   1:  PR[GP1:91,1] = PR[GP1:90,1] + 33.755;
   1:  PR[GP1:91,2] = PR[GP1:90,2] + -35.847;
   1:L PR[91] 10mm/sec CNT100;
   1:  PR[GP1:91,1] = PR[GP1:90,1] + 35.129;
   1:  PR[GP1:91,2] = PR[GP1:90,2] + -34.570;
   1:L PR[91] 10mm/sec CNT100;
   1:  PR[GP1:91,1] = PR[GP1:90,1] + 42.615;
   1:  PR[GP1:91,2] = PR[GP1:90,2] + -25.553;
   1:L PR[91] 10mm/sec CNT100;
   1:  PR[GP1:91,1] = PR[GP1:90,1] + 43.534;
   1:  PR[GP1:91,2] = PR[GP1:90,2] + -23.862;
   1:L PR[91] 10mm/sec CNT100;
   1:  PR[GP1:91,1] = PR[GP1:90,1] + 48.248;
   1:  PR[GP1:91,2] = PR[GP1:90,2] + -13.184;
   1:L PR[91] 10mm/sec CNT100;
   1:  PR[GP1:91,1] = PR[GP1:90,1] + 48.569;
   1:  PR[GP1:91,2] = PR[GP1:90,2] + -11.273;
   1:L PR[91] 10mm/sec CNT100;
   1:  PR[GP1:91,1] = PR[GP1:90,1] + 50.173;
   1:  PR[GP1:91,2] = PR[GP1:90,2] + 0.271;
   1:L PR[91] 10mm/sec CNT100;
   1:  PR[GP1:91,1] = PR[GP1:90,1] + 49.858;
   1:  PR[GP1:91,2] = PR[GP1:90,2] + 2.169;
   1:L PR[91] 10mm/sec CNT100;
   1:  PR[GP1:91,1] = PR[GP1:90,1] + 48.243;
   1:  PR[GP1:91,2] = PR[GP1:90,2] + 13.754;
   1:L PR[91] 10mm/sec CNT100;
   1:  PR[GP1:91,1] = PR[GP1:90,1] + 43.532;
   1:  PR[GP1:91,2] = PR[GP1:90,2] + 24.424;
   1:L PR[91] 10mm/sec CNT100;
   1:  PR[GP1:91,1] = PR[GP1:90,1] + 42.610;
   1:  PR[GP1:91,2] = PR[GP1:90,2] + 26.118;
   1:L PR[91] 10mm/sec CNT100;
   1:  PR[GP1:91,1] = PR[GP1:90,1] + 35.124;
   1:  PR[GP1:91,2] = PR[GP1:90,2] + 35.135;
   1:L PR[91] 10mm/sec CNT100;
   1:  PR[GP1:91,1] = PR[GP1:90,1] + 33.745;
   1:  PR[GP1:91,2] = PR[GP1:90,2] + 36.412;
   1:L PR[91] 10mm/sec CNT100;
   1:  PR[GP1:91,1] = PR[GP1:90,1] + 20.382;
   1:  PR[GP1:91,2] = PR[GP1:90,2] + 44.688;
   1:L PR[91] 10mm/sec CNT100;
   1:  PR[GP1:91,1] = PR[GP1:90,1] + 18.719;
   1:  PR[GP1:91,2] = PR[GP1:90,2] + 45.443;
   1:L PR[91] 10mm/sec CNT100;
   1:  PR[GP1:91,1] = PR[GP1:90,1] + 3.168;
   1:  PR[GP1:91,2] = PR[GP1:90,2] + 48.349;
   1:L PR[91] 10mm/sec CNT100;
   1:  PR[GP1:91,1] = PR[GP1:90,1] + 1.407;
   1:  PR[GP1:91,2] = PR[GP1:90,2] + 48.537;
   1:L PR[91] 10mm/sec CNT100;
   1:  PR[GP1:91,1] = PR[GP1:90,1] + -0.266;
   1:  PR[GP1:91,2] = PR[GP1:90,2] + 48.243;
   1:L PR[91] 10mm/sec CNT100;
   1:  PR[GP1:91,1] = PR[GP1:90,1] + -1.940;
   1:  PR[GP1:91,2] = PR[GP1:90,2] + 48.537;
   1:L PR[91] 10mm/sec CNT100;
   1:  PR[GP1:91,1] = PR[GP1:90,1] + -3.702;
   1:  PR[GP1:91,2] = PR[GP1:90,2] + 48.349;
   1:L PR[91] 10mm/sec CNT100;
   1:  PR[GP1:91,1] = PR[GP1:90,1] + -19.248;
   1:  PR[GP1:91,2] = PR[GP1:90,2] + 45.442;
   1:L PR[91] 10mm/sec CNT100;
   1:  PR[GP1:91,1] = PR[GP1:90,1] + -20.911;
   1:  PR[GP1:91,2] = PR[GP1:90,2] + 44.687;
   1:L PR[91] 10mm/sec CNT100;
   1:  PR[GP1:91,1] = PR[GP1:90,1] + -34.271;
   1:  PR[GP1:91,2] = PR[GP1:90,2] + 36.412;
   1:L PR[91] 10mm/sec CNT100;
   1:  PR[GP1:91,1] = PR[GP1:90,1] + -35.649;
   1:  PR[GP1:91,2] = PR[GP1:90,2] + 35.137;
   1:L PR[91] 10mm/sec CNT100;
   1:  PR[GP1:91,1] = PR[GP1:90,1] + -43.135;
   1:  PR[GP1:91,2] = PR[GP1:90,2] + 26.120;
   1:L PR[91] 10mm/sec CNT100;
   1:  PR[GP1:91,1] = PR[GP1:90,1] + -44.058;
   1:  PR[GP1:91,2] = PR[GP1:90,2] + 24.423;
   1:L PR[91] 10mm/sec CNT100;
   1:  PR[GP1:91,1] = PR[GP1:90,1] + -48.772;
   1:  PR[GP1:91,2] = PR[GP1:90,2] + 13.745;
   1:L PR[91] 10mm/sec CNT100;
   1:  PR[GP1:91,1] = PR[GP1:90,1] + -49.096;
   1:  PR[GP1:91,2] = PR[GP1:90,2] + 11.782;
   1:L PR[91] 10mm/sec CNT100;
   1:  PR[GP1:91,1] = PR[GP1:90,1] + -50.699;
   1:  PR[GP1:91,2] = PR[GP1:90,2] + 0.287;
   1:L PR[91] 10mm/sec CNT100;
   1:  PR[GP1:91,1] = PR[GP1:90,1] + -50.386;
   1:  PR[GP1:91,2] = PR[GP1:90,2] + -1.605;
   1:L PR[91] 10mm/sec CNT100;
   1:  PR[GP1:91,1] = PR[GP1:90,1] + -48.770;
   1:  PR[GP1:91,2] = PR[GP1:90,2] + -13.190;
   1:L PR[91] 10mm/sec CNT100;
   1:  PR[GP1:91,1] = PR[GP1:90,1] + -44.059;
   1:  PR[GP1:91,2] = PR[GP1:90,2] + -23.861;
   1:L PR[91] 10mm/sec CNT100;
   1:  PR[GP1:91,1] = PR[GP1:90,1] + -43.140;
   1:  PR[GP1:91,2] = PR[GP1:90,2] + -25.555;
   1:L PR[91] 10mm/sec CNT100;
   1:  PR[GP1:91,1] = PR[GP1:90,1] + -35.654;
   1:  PR[GP1:91,2] = PR[GP1:90,2] + -34.572;
   1:L PR[91] 10mm/sec CNT100;
   1:  PR[GP1:91,1] = PR[GP1:90,1] + -34.281;
   1:  PR[GP1:91,2] = PR[GP1:90,2] + -35.848;
   1:L PR[91] 10mm/sec CNT100;
   1:  PR[GP1:91,1] = PR[GP1:90,1] + -20.921;
   1:  PR[GP1:91,2] = PR[GP1:90,2] + -44.122;
   1:L PR[91] 10mm/sec CNT100;
   1:  PR[GP1:91,1] = PR[GP1:90,1] + -19.263;
   1:  PR[GP1:91,2] = PR[GP1:90,2] + -44.880;
   1:L PR[91] 10mm/sec CNT100;
   1:  PR[GP1:91,1] = PR[GP1:90,1] + -3.717;
   1:  PR[GP1:91,2] = PR[GP1:90,2] + -47.787;
   1:L PR[91] 10mm/sec CNT100;
   1:  PR[GP1:91,1] = PR[GP1:90,1] + -1.956;
   1:  PR[GP1:91,2] = PR[GP1:90,2] + -47.980;
   1:L PR[91] 10mm/sec CNT100;
   1:  PR[GP1:91,1] = PR[GP1:90,1] + -0.266;
   1:  PR[GP1:91,2] = PR[GP1:90,2] + -47.697;
   1:L PR[91] 10mm/sec CNT100;
   1:  PR[GP1:91,1] = PR[GP1:90,1] + 1.234;
   1:  PR[GP1:91,2] = PR[GP1:90,2] + -48.109;
   1:  PR[GP1:91,3] = PR[GP1:90,3] + 123.525;
   1:L PR[91] 10mm/sec CNT100;
   1:  PR[GP1:91,1] = PR[GP1:90,1] + 2.783;
   1:  PR[GP1:91,2] = PR[GP1:90,2] + -47.939;
   1:L PR[91] 10mm/sec CNT100;
   1:  PR[GP1:91,1] = PR[GP1:90,1] + 18.608;
   1:  PR[GP1:91,2] = PR[GP1:90,2] + -44.981;
   1:L PR[91] 10mm/sec CNT100;
   1:  PR[GP1:91,1] = PR[GP1:90,1] + 20.067;
   1:  PR[GP1:91,2] = PR[GP1:90,2] + -44.315;
   1:L PR[91] 10mm/sec CNT100;
   1:  PR[GP1:91,1] = PR[GP1:90,1] + 33.677;
   1:  PR[GP1:91,2] = PR[GP1:90,2] + -35.886;
   1:L PR[91] 10mm/sec CNT100;
   1:  PR[GP1:91,1] = PR[GP1:90,1] + 34.888;
   1:  PR[GP1:91,2] = PR[GP1:90,2] + -34.760;
   1:L PR[91] 10mm/sec CNT100;
   1:  PR[GP1:91,1] = PR[GP1:90,1] + 42.517;
   1:  PR[GP1:91,2] = PR[GP1:90,2] + -25.570;
   1:L PR[91] 10mm/sec CNT100;
   1:  PR[GP1:91,1] = PR[GP1:90,1] + 43.328;
   1:  PR[GP1:91,2] = PR[GP1:90,2] + -24.078;
   1:L PR[91] 10mm/sec CNT100;
   1:  PR[GP1:91,1] = PR[GP1:90,1] + 48.135;
   1:  PR[GP1:91,2] = PR[GP1:90,2] + -13.189;
   1:L PR[91] 10mm/sec CNT100;
   1:  PR[GP1:91,1] = PR[GP1:90,1] + 48.418;
   1:  PR[GP1:91,2] = PR[GP1:90,2] + -11.503;
   1:L PR[91] 10mm/sec CNT100;
   1:  PR[GP1:91,1] = PR[GP1:90,1] + 50.055;
   1:  PR[GP1:91,2] = PR[GP1:90,2] + 0.271;
   1:L PR[91] 10mm/sec CNT100;
   1:  PR[GP1:91,1] = PR[GP1:90,1] + 49.778;
   1:  PR[GP1:91,2] = PR[GP1:90,2] + 1.945;
   1:L PR[91] 10mm/sec CNT100;
   1:  PR[GP1:91,1] = PR[GP1:90,1] + 48.130;
   1:  PR[GP1:91,2] = PR[GP1:90,2] + 13.759;
   1:L PR[91] 10mm/sec CNT100;
   1:  PR[GP1:91,1] = PR[GP1:90,1] + 43.326;
   1:  PR[GP1:91,2] = PR[GP1:90,2] + 24.640;
   1:L PR[91] 10mm/sec CNT100;
   1:  PR[GP1:91,1] = PR[GP1:90,1] + 42.512;
   1:  PR[GP1:91,2] = PR[GP1:90,2] + 26.134;
   1:L PR[91] 10mm/sec CNT100;
   1:  PR[GP1:91,1] = PR[GP1:90,1] + 34.883;
   1:  PR[GP1:91,2] = PR[GP1:90,2] + 35.324;
   1:L PR[91] 10mm/sec CNT100;
   1:  PR[GP1:91,1] = PR[GP1:90,1] + 33.668;
   1:  PR[GP1:91,2] = PR[GP1:90,2] + 36.450;
   1:L PR[91] 10mm/sec CNT100;
   1:  PR[GP1:91,1] = PR[GP1:90,1] + 20.058;
   1:  PR[GP1:91,2] = PR[GP1:90,2] + 44.879;
   1:L PR[91] 10mm/sec CNT100;
   1:  PR[GP1:91,1] = PR[GP1:90,1] + 18.595;
   1:  PR[GP1:91,2] = PR[GP1:90,2] + 45.542;
   1:L PR[91] 10mm/sec CNT100;
   1:  PR[GP1:91,1] = PR[GP1:90,1] + 2.769;
   1:  PR[GP1:91,2] = PR[GP1:90,2] + 48.500;
   1:L PR[91] 10mm/sec CNT100;
   1:  PR[GP1:91,1] = PR[GP1:90,1] + 1.220;
   1:  PR[GP1:91,2] = PR[GP1:90,2] + 48.666;
   1:L PR[91] 10mm/sec CNT100;
   1:  PR[GP1:91,1] = PR[GP1:90,1] + -0.266;
   1:  PR[GP1:91,2] = PR[GP1:90,2] + 48.405;
   1:L PR[91] 10mm/sec CNT100;
   1:  PR[GP1:91,1] = PR[GP1:90,1] + -1.753;
   1:  PR[GP1:91,2] = PR[GP1:90,2] + 48.666;
   1:L PR[91] 10mm/sec CNT100;
   1:  PR[GP1:91,1] = PR[GP1:90,1] + -3.303;
   1:  PR[GP1:91,2] = PR[GP1:90,2] + 48.501;
   1:L PR[91] 10mm/sec CNT100;
   1:  PR[GP1:91,1] = PR[GP1:90,1] + -19.124;
   1:  PR[GP1:91,2] = PR[GP1:90,2] + 45.542;
   1:L PR[91] 10mm/sec CNT100;
   1:  PR[GP1:91,1] = PR[GP1:90,1] + -20.587;
   1:  PR[GP1:91,2] = PR[GP1:90,2] + 44.877;
   1:L PR[91] 10mm/sec CNT100;
   1:  PR[GP1:91,1] = PR[GP1:90,1] + -34.193;
   1:  PR[GP1:91,2] = PR[GP1:90,2] + 36.450;
   1:L PR[91] 10mm/sec CNT100;
   1:  PR[GP1:91,1] = PR[GP1:90,1] + -35.408;
   1:  PR[GP1:91,2] = PR[GP1:90,2] + 35.326;
   1:L PR[91] 10mm/sec CNT100;
   1:  PR[GP1:91,1] = PR[GP1:90,1] + -43.038;
   1:  PR[GP1:91,2] = PR[GP1:90,2] + 26.136;
   1:L PR[91] 10mm/sec CNT100;
   1:  PR[GP1:91,1] = PR[GP1:90,1] + -43.852;
   1:  PR[GP1:91,2] = PR[GP1:90,2] + 24.639;
   1:L PR[91] 10mm/sec CNT100;
   1:  PR[GP1:91,1] = PR[GP1:90,1] + -48.659;
   1:  PR[GP1:91,2] = PR[GP1:90,2] + 13.750;
   1:L PR[91] 10mm/sec CNT100;
   1:  PR[GP1:91,1] = PR[GP1:90,1] + -48.945;
   1:  PR[GP1:91,2] = PR[GP1:90,2] + 12.018;
   1:L PR[91] 10mm/sec CNT100;
   1:  PR[GP1:91,1] = PR[GP1:90,1] + -50.581;
   1:  PR[GP1:91,2] = PR[GP1:90,2] + 0.287;
   1:L PR[91] 10mm/sec CNT100;
   1:  PR[GP1:91,1] = PR[GP1:90,1] + -50.305;
   1:  PR[GP1:91,2] = PR[GP1:90,2] + -1.382;
   1:L PR[91] 10mm/sec CNT100;
   1:  PR[GP1:91,1] = PR[GP1:90,1] + -48.657;
   1:  PR[GP1:91,2] = PR[GP1:90,2] + -13.195;
   1:L PR[91] 10mm/sec CNT100;
   1:  PR[GP1:91,1] = PR[GP1:90,1] + -43.853;
   1:  PR[GP1:91,2] = PR[GP1:90,2] + -24.077;
   1:L PR[91] 10mm/sec CNT100;
   1:  PR[GP1:91,1] = PR[GP1:90,1] + -43.043;
   1:  PR[GP1:91,2] = PR[GP1:90,2] + -25.572;
   1:L PR[91] 10mm/sec CNT100;
   1:  PR[GP1:91,1] = PR[GP1:90,1] + -35.412;
   1:  PR[GP1:91,2] = PR[GP1:90,2] + -34.763;
   1:L PR[91] 10mm/sec CNT100;
   1:  PR[GP1:91,1] = PR[GP1:90,1] + -34.202;
   1:  PR[GP1:91,2] = PR[GP1:90,2] + -35.886;
   1:L PR[91] 10mm/sec CNT100;
   1:  PR[GP1:91,1] = PR[GP1:90,1] + -20.596;
   1:  PR[GP1:91,2] = PR[GP1:90,2] + -44.313;
   1:L PR[91] 10mm/sec CNT100;
   1:  PR[GP1:91,1] = PR[GP1:90,1] + -19.137;
   1:  PR[GP1:91,2] = PR[GP1:90,2] + -44.980;
   1:L PR[91] 10mm/sec CNT100;
   1:  PR[GP1:91,1] = PR[GP1:90,1] + -3.317;
   1:  PR[GP1:91,2] = PR[GP1:90,2] + -47.939;
   1:L PR[91] 10mm/sec CNT100;
   1:  PR[GP1:91,1] = PR[GP1:90,1] + -1.767;
   1:  PR[GP1:91,2] = PR[GP1:90,2] + -48.109;
   1:L PR[91] 10mm/sec CNT100;
   1:  PR[GP1:91,1] = PR[GP1:90,1] + -0.266;
   1:  PR[GP1:91,2] = PR[GP1:90,2] + -47.857;
   1:L PR[91] 10mm/sec CNT100;
   1:  PR[GP1:91,1] = PR[GP1:90,1] + 1.044;
   1:  PR[GP1:91,2] = PR[GP1:90,2] + -48.237;
   1:  PR[GP1:91,3] = PR[GP1:90,3] + 124.135;
   1:L PR[91] 10mm/sec CNT100;
   1:  PR[GP1:91,1] = PR[GP1:90,1] + 2.382;
   1:  PR[GP1:91,2] = PR[GP1:90,2] + -48.090;
   1:L PR[91] 10mm/sec CNT100;
   1:  PR[GP1:91,1] = PR[GP1:90,1] + 18.482;
   1:  PR[GP1:91,2] = PR[GP1:90,2] + -45.081;
   1:L PR[91] 10mm/sec CNT100;
   1:  PR[GP1:91,1] = PR[GP1:90,1] + 19.742;
   1:  PR[GP1:91,2] = PR[GP1:90,2] + -44.506;
   1:L PR[91] 10mm/sec CNT100;
   1:  PR[GP1:91,1] = PR[GP1:90,1] + 33.599;
   1:  PR[GP1:91,2] = PR[GP1:90,2] + -35.924;
   1:L PR[91] 10mm/sec CNT100;
   1:  PR[GP1:91,1] = PR[GP1:90,1] + 34.646;
   1:  PR[GP1:91,2] = PR[GP1:90,2] + -34.951;
   1:L PR[91] 10mm/sec CNT100;
   1:  PR[GP1:91,1] = PR[GP1:90,1] + 42.419;
   1:  PR[GP1:91,2] = PR[GP1:90,2] + -25.586;
   1:L PR[91] 10mm/sec CNT100;
   1:  PR[GP1:91,1] = PR[GP1:90,1] + 43.121;
   1:  PR[GP1:91,2] = PR[GP1:90,2] + -24.295;
   1:L PR[91] 10mm/sec CNT100;
   1:  PR[GP1:91,1] = PR[GP1:90,1] + 48.022;
   1:  PR[GP1:91,2] = PR[GP1:90,2] + -13.194;
   1:L PR[91] 10mm/sec CNT100;
   1:  PR[GP1:91,1] = PR[GP1:90,1] + 48.267;
   1:  PR[GP1:91,2] = PR[GP1:90,2] + -11.734;
   1:L PR[91] 10mm/sec CNT100;
   1:  PR[GP1:91,1] = PR[GP1:90,1] + 49.937;
   1:  PR[GP1:91,2] = PR[GP1:90,2] + 0.271;
   1:L PR[91] 10mm/sec CNT100;
   1:  PR[GP1:91,1] = PR[GP1:90,1] + 49.697;
   1:  PR[GP1:91,2] = PR[GP1:90,2] + 1.721;
   1:L PR[91] 10mm/sec CNT100;
   1:  PR[GP1:91,1] = PR[GP1:90,1] + 48.017;
   1:  PR[GP1:91,2] = PR[GP1:90,2] + 13.763;
   1:L PR[91] 10mm/sec CNT100;
   1:  PR[GP1:91,1] = PR[GP1:90,1] + 43.120;
   1:  PR[GP1:91,2] = PR[GP1:90,2] + 24.856;
   1:L PR[91] 10mm/sec CNT100;
   1:  PR[GP1:91,1] = PR[GP1:90,1] + 42.415;
   1:  PR[GP1:91,2] = PR[GP1:90,2] + 26.149;
   1:L PR[91] 10mm/sec CNT100;
   1:  PR[GP1:91,1] = PR[GP1:90,1] + 34.642;
   1:  PR[GP1:91,2] = PR[GP1:90,2] + 35.514;
   1:L PR[91] 10mm/sec CNT100;
   1:  PR[GP1:91,1] = PR[GP1:90,1] + 33.591;
   1:  PR[GP1:91,2] = PR[GP1:90,2] + 36.487;
   1:L PR[91] 10mm/sec CNT100;
   1:  PR[GP1:91,1] = PR[GP1:90,1] + 19.734;
   1:  PR[GP1:91,2] = PR[GP1:90,2] + 45.069;
   1:L PR[91] 10mm/sec CNT100;
   1:  PR[GP1:91,1] = PR[GP1:90,1] + 18.470;
   1:  PR[GP1:91,2] = PR[GP1:90,2] + 45.642;
   1:L PR[91] 10mm/sec CNT100;
   1:  PR[GP1:91,1] = PR[GP1:90,1] + 2.371;
   1:  PR[GP1:91,2] = PR[GP1:90,2] + 48.652;
   1:L PR[91] 10mm/sec CNT100;
   1:  PR[GP1:91,1] = PR[GP1:90,1] + 1.033;
   1:  PR[GP1:91,2] = PR[GP1:90,2] + 48.795;
   1:L PR[91] 10mm/sec CNT100;
   1:  PR[GP1:91,1] = PR[GP1:90,1] + -0.266;
   1:  PR[GP1:91,2] = PR[GP1:90,2] + 48.566;
   1:L PR[91] 10mm/sec CNT100;
   1:  PR[GP1:91,1] = PR[GP1:90,1] + -1.566;
   1:  PR[GP1:91,2] = PR[GP1:90,2] + 48.794;
   1:L PR[91] 10mm/sec CNT100;
   1:  PR[GP1:91,1] = PR[GP1:90,1] + -2.905;
   1:  PR[GP1:91,2] = PR[GP1:90,2] + 48.652;
   1:L PR[91] 10mm/sec CNT100;
   1:  PR[GP1:91,1] = PR[GP1:90,1] + -19.000;
   1:  PR[GP1:91,2] = PR[GP1:90,2] + 45.641;
   1:L PR[91] 10mm/sec CNT100;
   1:  PR[GP1:91,1] = PR[GP1:90,1] + -20.263;
   1:  PR[GP1:91,2] = PR[GP1:90,2] + 45.068;
   1:L PR[91] 10mm/sec CNT100;
   1:  PR[GP1:91,1] = PR[GP1:90,1] + -34.116;
   1:  PR[GP1:91,2] = PR[GP1:90,2] + 36.488;
   1:L PR[91] 10mm/sec CNT100;
   1:  PR[GP1:91,1] = PR[GP1:90,1] + -35.166;
   1:  PR[GP1:91,2] = PR[GP1:90,2] + 35.516;
   1:L PR[91] 10mm/sec CNT100;
   1:  PR[GP1:91,1] = PR[GP1:90,1] + -42.941;
   1:  PR[GP1:91,2] = PR[GP1:90,2] + 26.151;
   1:L PR[91] 10mm/sec CNT100;
   1:  PR[GP1:91,1] = PR[GP1:90,1] + -43.646;
   1:  PR[GP1:91,2] = PR[GP1:90,2] + 24.855;
   1:L PR[91] 10mm/sec CNT100;
   1:  PR[GP1:91,1] = PR[GP1:90,1] + -48.546;
   1:  PR[GP1:91,2] = PR[GP1:90,2] + 13.755;
   1:L PR[91] 10mm/sec CNT100;
   1:  PR[GP1:91,1] = PR[GP1:90,1] + -48.794;
   1:  PR[GP1:91,2] = PR[GP1:90,2] + 12.255;
   1:L PR[91] 10mm/sec CNT100;
   1:  PR[GP1:91,1] = PR[GP1:90,1] + -50.463;
   1:  PR[GP1:91,2] = PR[GP1:90,2] + 0.287;
   1:L PR[91] 10mm/sec CNT100;
   1:  PR[GP1:91,1] = PR[GP1:90,1] + -50.224;
   1:  PR[GP1:91,2] = PR[GP1:90,2] + -1.158;
   1:L PR[91] 10mm/sec CNT100;
   1:  PR[GP1:91,1] = PR[GP1:90,1] + -48.544;
   1:  PR[GP1:91,2] = PR[GP1:90,2] + -13.201;
   1:L PR[91] 10mm/sec CNT100;
   1:  PR[GP1:91,1] = PR[GP1:90,1] + -43.647;
   1:  PR[GP1:91,2] = PR[GP1:90,2] + -24.294;
   1:L PR[91] 10mm/sec CNT100;
   1:  PR[GP1:91,1] = PR[GP1:90,1] + -42.945;
   1:  PR[GP1:91,2] = PR[GP1:90,2] + -25.588;
   1:L PR[91] 10mm/sec CNT100;
   1:  PR[GP1:91,1] = PR[GP1:90,1] + -35.170;
   1:  PR[GP1:91,2] = PR[GP1:90,2] + -34.953;
   1:L PR[91] 10mm/sec CNT100;
   1:  PR[GP1:91,1] = PR[GP1:90,1] + -34.124;
   1:  PR[GP1:91,2] = PR[GP1:90,2] + -35.925;
   1:L PR[91] 10mm/sec CNT100;
   1:  PR[GP1:91,1] = PR[GP1:90,1] + -20.271;
   1:  PR[GP1:91,2] = PR[GP1:90,2] + -44.505;
   1:L PR[91] 10mm/sec CNT100;
   1:  PR[GP1:91,1] = PR[GP1:90,1] + -19.011;
   1:  PR[GP1:91,2] = PR[GP1:90,2] + -45.080;
   1:L PR[91] 10mm/sec CNT100;
   1:  PR[GP1:91,1] = PR[GP1:90,1] + -2.916;
   1:  PR[GP1:91,2] = PR[GP1:90,2] + -48.090;
   1:L PR[91] 10mm/sec CNT100;
   1:  PR[GP1:91,1] = PR[GP1:90,1] + -1.578;
   1:  PR[GP1:91,2] = PR[GP1:90,2] + -48.237;
   1:L PR[91] 10mm/sec CNT100;
   1:  PR[GP1:91,1] = PR[GP1:90,1] + -0.266;
   1:  PR[GP1:91,2] = PR[GP1:90,2] + -48.017;
   1:L PR[91] 10mm/sec CNT100;
   1:  PR[GP1:91,1] = PR[GP1:90,1] + 0.855;
   1:  PR[GP1:91,2] = PR[GP1:90,2] + -48.366;
   1:  PR[GP1:91,3] = PR[GP1:90,3] + 124.745;
   1:L PR[91] 10mm/sec CNT100;
   1:  PR[GP1:91,1] = PR[GP1:90,1] + 1.982;
   1:  PR[GP1:91,2] = PR[GP1:90,2] + -48.242;
   1:L PR[91] 10mm/sec CNT100;
   1:  PR[GP1:91,1] = PR[GP1:90,1] + 18.355;
   1:  PR[GP1:91,2] = PR[GP1:90,2] + -45.182;
   1:L PR[91] 10mm/sec CNT100;
   1:  PR[GP1:91,1] = PR[GP1:90,1] + 19.416;
   1:  PR[GP1:91,2] = PR[GP1:90,2] + -44.697;
   1:L PR[91] 10mm/sec CNT100;
   1:  PR[GP1:91,1] = PR[GP1:90,1] + 33.520;
   1:  PR[GP1:91,2] = PR[GP1:90,2] + -35.962;
   1:L PR[91] 10mm/sec CNT100;
   1:  PR[GP1:91,1] = PR[GP1:90,1] + 34.404;
   1:  PR[GP1:91,2] = PR[GP1:90,2] + -35.141;
   1:L PR[91] 10mm/sec CNT100;
   1:  PR[GP1:91,1] = PR[GP1:90,1] + 42.321;
   1:  PR[GP1:91,2] = PR[GP1:90,2] + -25.603;
   1:L PR[91] 10mm/sec CNT100;
   1:  PR[GP1:91,1] = PR[GP1:90,1] + 42.915;
   1:  PR[GP1:91,2] = PR[GP1:90,2] + -24.511;
   1:L PR[91] 10mm/sec CNT100;
   1:  PR[GP1:91,1] = PR[GP1:90,1] + 47.909;
   1:  PR[GP1:91,2] = PR[GP1:90,2] + -13.199;
   1:L PR[91] 10mm/sec CNT100;
   1:  PR[GP1:91,1] = PR[GP1:90,1] + 48.116;
   1:  PR[GP1:91,2] = PR[GP1:90,2] + -11.965;
   1:L PR[91] 10mm/sec CNT100;
   1:  PR[GP1:91,1] = PR[GP1:90,1] + 49.819;
   1:  PR[GP1:91,2] = PR[GP1:90,2] + 0.271;
   1:L PR[91] 10mm/sec CNT100;
   1:  PR[GP1:91,1] = PR[GP1:90,1] + 49.616;
   1:  PR[GP1:91,2] = PR[GP1:90,2] + 1.497;
   1:L PR[91] 10mm/sec CNT100;
   1:  PR[GP1:91,1] = PR[GP1:90,1] + 47.904;
   1:  PR[GP1:91,2] = PR[GP1:90,2] + 13.768;
   1:L PR[91] 10mm/sec CNT100;
   1:  PR[GP1:91,1] = PR[GP1:90,1] + 42.914;
   1:  PR[GP1:91,2] = PR[GP1:90,2] + 25.071;
   1:L PR[91] 10mm/sec CNT100;
   1:  PR[GP1:91,1] = PR[GP1:90,1] + 42.318;
   1:  PR[GP1:91,2] = PR[GP1:90,2] + 26.165;
   1:L PR[91] 10mm/sec CNT100;
   1:  PR[GP1:91,1] = PR[GP1:90,1] + 34.400;
   1:  PR[GP1:91,2] = PR[GP1:90,2] + 35.703;
   1:L PR[91] 10mm/sec CNT100;
   1:  PR[GP1:91,1] = PR[GP1:90,1] + 33.514;
   1:  PR[GP1:91,2] = PR[GP1:90,2] + 36.525;
   1:L PR[91] 10mm/sec CNT100;
   1:  PR[GP1:91,1] = PR[GP1:90,1] + 19.410;
   1:  PR[GP1:91,2] = PR[GP1:90,2] + 45.260;
   1:L PR[91] 10mm/sec CNT100;
   1:  PR[GP1:91,1] = PR[GP1:90,1] + 18.346;
   1:  PR[GP1:91,2] = PR[GP1:90,2] + 45.742;
   1:L PR[91] 10mm/sec CNT100;
   1:  PR[GP1:91,1] = PR[GP1:90,1] + 1.972;
   1:  PR[GP1:91,2] = PR[GP1:90,2] + 48.803;
   1:L PR[91] 10mm/sec CNT100;
   1:  PR[GP1:91,1] = PR[GP1:90,1] + 0.845;
   1:  PR[GP1:91,2] = PR[GP1:90,2] + 48.923;
   1:L PR[91] 10mm/sec CNT100;
   1:  PR[GP1:91,1] = PR[GP1:90,1] + -0.266;
   1:  PR[GP1:91,2] = PR[GP1:90,2] + 48.728;
   1:L PR[91] 10mm/sec CNT100;
   1:  PR[GP1:91,1] = PR[GP1:90,1] + -1.379;
   1:  PR[GP1:91,2] = PR[GP1:90,2] + 48.923;
   1:L PR[91] 10mm/sec CNT100;
   1:  PR[GP1:91,1] = PR[GP1:90,1] + -2.506;
   1:  PR[GP1:91,2] = PR[GP1:90,2] + 48.803;
   1:L PR[91] 10mm/sec CNT100;
   1:  PR[GP1:91,1] = PR[GP1:90,1] + -18.875;
   1:  PR[GP1:91,2] = PR[GP1:90,2] + 45.741;
   1:L PR[91] 10mm/sec CNT100;
   1:  PR[GP1:91,1] = PR[GP1:90,1] + -19.939;
   1:  PR[GP1:91,2] = PR[GP1:90,2] + 45.258;
   1:L PR[91] 10mm/sec CNT100;
   1:  PR[GP1:91,1] = PR[GP1:90,1] + -34.039;
   1:  PR[GP1:91,2] = PR[GP1:90,2] + 36.525;
   1:L PR[91] 10mm/sec CNT100;
   1:  PR[GP1:91,1] = PR[GP1:90,1] + -34.925;
   1:  PR[GP1:91,2] = PR[GP1:90,2] + 35.705;
   1:L PR[91] 10mm/sec CNT100;
   1:  PR[GP1:91,1] = PR[GP1:90,1] + -42.844;
   1:  PR[GP1:91,2] = PR[GP1:90,2] + 26.167;
   1:L PR[91] 10mm/sec CNT100;
   1:  PR[GP1:91,1] = PR[GP1:90,1] + -43.440;
   1:  PR[GP1:91,2] = PR[GP1:90,2] + 25.071;
   1:L PR[91] 10mm/sec CNT100;
   1:  PR[GP1:91,1] = PR[GP1:90,1] + -48.434;
   1:  PR[GP1:91,2] = PR[GP1:90,2] + 13.760;
   1:L PR[91] 10mm/sec CNT100;
   1:  PR[GP1:91,1] = PR[GP1:90,1] + -48.643;
   1:  PR[GP1:91,2] = PR[GP1:90,2] + 12.491;
   1:L PR[91] 10mm/sec CNT100;
   1:  PR[GP1:91,1] = PR[GP1:90,1] + -50.345;
   1:  PR[GP1:91,2] = PR[GP1:90,2] + 0.287;
   1:L PR[91] 10mm/sec CNT100;
   1:  PR[GP1:91,1] = PR[GP1:90,1] + -50.143;
   1:  PR[GP1:91,2] = PR[GP1:90,2] + -0.935;
   1:L PR[91] 10mm/sec CNT100;
   1:  PR[GP1:91,1] = PR[GP1:90,1] + -48.431;
   1:  PR[GP1:91,2] = PR[GP1:90,2] + -13.206;
   1:L PR[91] 10mm/sec CNT100;
   1:  PR[GP1:91,1] = PR[GP1:90,1] + -43.441;
   1:  PR[GP1:91,2] = PR[GP1:90,2] + -24.511;
   1:L PR[91] 10mm/sec CNT100;
   1:  PR[GP1:91,1] = PR[GP1:90,1] + -42.847;
   1:  PR[GP1:91,2] = PR[GP1:90,2] + -25.605;
   1:L PR[91] 10mm/sec CNT100;
   1:  PR[GP1:91,1] = PR[GP1:90,1] + -34.928;
   1:  PR[GP1:91,2] = PR[GP1:90,2] + -35.143;
   1:L PR[91] 10mm/sec CNT100;
   1:  PR[GP1:91,1] = PR[GP1:90,1] + -34.045;
   1:  PR[GP1:91,2] = PR[GP1:90,2] + -35.963;
   1:L PR[91] 10mm/sec CNT100;
   1:  PR[GP1:91,1] = PR[GP1:90,1] + -19.945;
   1:  PR[GP1:91,2] = PR[GP1:90,2] + -44.696;
   1:L PR[91] 10mm/sec CNT100;
   1:  PR[GP1:91,1] = PR[GP1:90,1] + -18.885;
   1:  PR[GP1:91,2] = PR[GP1:90,2] + -45.181;
   1:L PR[91] 10mm/sec CNT100;
   1:  PR[GP1:91,1] = PR[GP1:90,1] + -2.516;
   1:  PR[GP1:91,2] = PR[GP1:90,2] + -48.242;
   1:L PR[91] 10mm/sec CNT100;
   1:  PR[GP1:91,1] = PR[GP1:90,1] + -1.389;
   1:  PR[GP1:91,2] = PR[GP1:90,2] + -48.366;
   1:L PR[91] 10mm/sec CNT100;
   1:  PR[GP1:91,1] = PR[GP1:90,1] + -0.266;
   1:  PR[GP1:91,2] = PR[GP1:90,2] + -48.178;
   1:L PR[91] 10mm/sec CNT100;
   1:  PR[GP1:91,1] = PR[GP1:90,1] + 0.666;
   1:  PR[GP1:91,2] = PR[GP1:90,2] + -48.494;
   1:  PR[GP1:91,3] = PR[GP1:90,3] + 125.355;
   1:L PR[91] 10mm/sec CNT100;
   1:  PR[GP1:91,1] = PR[GP1:90,1] + 1.581;
   1:  PR[GP1:91,2] = PR[GP1:90,2] + -48.394;
   1:L PR[91] 10mm/sec CNT100;
   1:  PR[GP1:91,1] = PR[GP1:90,1] + 18.229;
   1:  PR[GP1:91,2] = PR[GP1:90,2] + -45.282;
   1:L PR[91] 10mm/sec CNT100;
   1:  PR[GP1:91,1] = PR[GP1:90,1] + 19.091;
   1:  PR[GP1:91,2] = PR[GP1:90,2] + -44.889;
   1:L PR[91] 10mm/sec CNT100;
   1:  PR[GP1:91,1] = PR[GP1:90,1] + 33.442;
   1:  PR[GP1:91,2] = PR[GP1:90,2] + -36.001;
   1:L PR[91] 10mm/sec CNT100;
   1:  PR[GP1:91,1] = PR[GP1:90,1] + 34.162;
   1:  PR[GP1:91,2] = PR[GP1:90,2] + -35.331;
   1:L PR[91] 10mm/sec CNT100;
   1:  PR[GP1:91,1] = PR[GP1:90,1] + 42.224;
   1:  PR[GP1:91,2] = PR[GP1:90,2] + -25.620;
   1:L PR[91] 10mm/sec CNT100;
   1:  PR[GP1:91,1] = PR[GP1:90,1] + 42.709;
   1:  PR[GP1:91,2] = PR[GP1:90,2] + -24.727;
   1:L PR[91] 10mm/sec CNT100;
   1:  PR[GP1:91,1] = PR[GP1:90,1] + 47.796;
   1:  PR[GP1:91,2] = PR[GP1:90,2] + -13.204;
   1:L PR[91] 10mm/sec CNT100;
   1:  PR[GP1:91,1] = PR[GP1:90,1] + 47.965;
   1:  PR[GP1:91,2] = PR[GP1:90,2] + -12.195;
   1:L PR[91] 10mm/sec CNT100;
   1:  PR[GP1:91,1] = PR[GP1:90,1] + 49.701;
   1:  PR[GP1:91,2] = PR[GP1:90,2] + 0.271;
   1:L PR[91] 10mm/sec CNT100;
   1:  PR[GP1:91,1] = PR[GP1:90,1] + 49.535;
   1:  PR[GP1:91,2] = PR[GP1:90,2] + 1.273;
   1:L PR[91] 10mm/sec CNT100;
   1:  PR[GP1:91,1] = PR[GP1:90,1] + 47.792;
   1:  PR[GP1:91,2] = PR[GP1:90,2] + 13.772;
   1:L PR[91] 10mm/sec CNT100;
   1:  PR[GP1:91,1] = PR[GP1:90,1] + 42.708;
   1:  PR[GP1:91,2] = PR[GP1:90,2] + 25.287;
   1:L PR[91] 10mm/sec CNT100;
   1:  PR[GP1:91,1] = PR[GP1:90,1] + 42.221;
   1:  PR[GP1:91,2] = PR[GP1:90,2] + 26.181;
   1:L PR[91] 10mm/sec CNT100;
   1:  PR[GP1:91,1] = PR[GP1:90,1] + 34.159;
   1:  PR[GP1:91,2] = PR[GP1:90,2] + 35.893;
   1:L PR[91] 10mm/sec CNT100;
   1:  PR[GP1:91,1] = PR[GP1:90,1] + 33.437;
   1:  PR[GP1:91,2] = PR[GP1:90,2] + 36.562;
   1:L PR[91] 10mm/sec CNT100;
   1:  PR[GP1:91,1] = PR[GP1:90,1] + 19.086;
   1:  PR[GP1:91,2] = PR[GP1:90,2] + 45.450;
   1:L PR[91] 10mm/sec CNT100;
   1:  PR[GP1:91,1] = PR[GP1:90,1] + 18.221;
   1:  PR[GP1:91,2] = PR[GP1:90,2] + 45.842;
   1:L PR[91] 10mm/sec CNT100;
   1:  PR[GP1:91,1] = PR[GP1:90,1] + 1.573;
   1:  PR[GP1:91,2] = PR[GP1:90,2] + 48.954;
   1:L PR[91] 10mm/sec CNT100;
   1:  PR[GP1:91,1] = PR[GP1:90,1] + 0.658;
   1:  PR[GP1:91,2] = PR[GP1:90,2] + 49.052;
   1:L PR[91] 10mm/sec CNT100;
   1:  PR[GP1:91,1] = PR[GP1:90,1] + -0.266;
   1:  PR[GP1:91,2] = PR[GP1:90,2] + 48.889;
   1:L PR[91] 10mm/sec CNT100;
   1:  PR[GP1:91,1] = PR[GP1:90,1] + -1.192;
   1:  PR[GP1:91,2] = PR[GP1:90,2] + 49.052;
   1:L PR[91] 10mm/sec CNT100;
   1:  PR[GP1:91,1] = PR[GP1:90,1] + -2.108;
   1:  PR[GP1:91,2] = PR[GP1:90,2] + 48.954;
   1:L PR[91] 10mm/sec CNT100;
   1:  PR[GP1:91,1] = PR[GP1:90,1] + -18.751;
   1:  PR[GP1:91,2] = PR[GP1:90,2] + 45.841;
   1:L PR[91] 10mm/sec CNT100;
   1:  PR[GP1:91,1] = PR[GP1:90,1] + -19.615;
   1:  PR[GP1:91,2] = PR[GP1:90,2] + 45.449;
   1:L PR[91] 10mm/sec CNT100;
   1:  PR[GP1:91,1] = PR[GP1:90,1] + -33.962;
   1:  PR[GP1:91,2] = PR[GP1:90,2] + 36.563;
   1:L PR[91] 10mm/sec CNT100;
   1:  PR[GP1:91,1] = PR[GP1:90,1] + -34.684;
   1:  PR[GP1:91,2] = PR[GP1:90,2] + 35.895;
   1:L PR[91] 10mm/sec CNT100;
   1:  PR[GP1:91,1] = PR[GP1:90,1] + -42.747;
   1:  PR[GP1:91,2] = PR[GP1:90,2] + 26.183;
   1:L PR[91] 10mm/sec CNT100;
   1:  PR[GP1:91,1] = PR[GP1:90,1] + -43.234;
   1:  PR[GP1:91,2] = PR[GP1:90,2] + 25.287;
   1:L PR[91] 10mm/sec CNT100;
   1:  PR[GP1:91,1] = PR[GP1:90,1] + -48.321;
   1:  PR[GP1:91,2] = PR[GP1:90,2] + 13.765;
   1:L PR[91] 10mm/sec CNT100;
   1:  PR[GP1:91,1] = PR[GP1:90,1] + -48.492;
   1:  PR[GP1:91,2] = PR[GP1:90,2] + 12.727;
   1:L PR[91] 10mm/sec CNT100;
   1:  PR[GP1:91,1] = PR[GP1:90,1] + -50.227;
   1:  PR[GP1:91,2] = PR[GP1:90,2] + 0.287;
   1:L PR[91] 10mm/sec CNT100;
   1:  PR[GP1:91,1] = PR[GP1:90,1] + -50.062;
   1:  PR[GP1:91,2] = PR[GP1:90,2] + -0.711;
   1:L PR[91] 10mm/sec CNT100;
   1:  PR[GP1:91,1] = PR[GP1:90,1] + -48.319;
   1:  PR[GP1:91,2] = PR[GP1:90,2] + -13.211;
   1:L PR[91] 10mm/sec CNT100;
   1:  PR[GP1:91,1] = PR[GP1:90,1] + -43.235;
   1:  PR[GP1:91,2] = PR[GP1:90,2] + -24.727;
   1:L PR[91] 10mm/sec CNT100;
   1:  PR[GP1:91,1] = PR[GP1:90,1] + -42.749;
   1:  PR[GP1:91,2] = PR[GP1:90,2] + -25.621;
   1:L PR[91] 10mm/sec CNT100;
   1:  PR[GP1:91,1] = PR[GP1:90,1] + -34.686;
   1:  PR[GP1:91,2] = PR[GP1:90,2] + -35.333;
   1:L PR[91] 10mm/sec CNT100;
   1:  PR[GP1:91,1] = PR[GP1:90,1] + -33.967;
   1:  PR[GP1:91,2] = PR[GP1:90,2] + -36.001;
   1:L PR[91] 10mm/sec CNT100;
   1:  PR[GP1:91,1] = PR[GP1:90,1] + -19.620;
   1:  PR[GP1:91,2] = PR[GP1:90,2] + -44.887;
   1:L PR[91] 10mm/sec CNT100;
   1:  PR[GP1:91,1] = PR[GP1:90,1] + -18.758;
   1:  PR[GP1:91,2] = PR[GP1:90,2] + -45.281;
   1:L PR[91] 10mm/sec CNT100;
   1:  PR[GP1:91,1] = PR[GP1:90,1] + -2.116;
   1:  PR[GP1:91,2] = PR[GP1:90,2] + -48.394;
   1:L PR[91] 10mm/sec CNT100;
   1:  PR[GP1:91,1] = PR[GP1:90,1] + -1.200;
   1:  PR[GP1:91,2] = PR[GP1:90,2] + -48.494;
   1:L PR[91] 10mm/sec CNT100;
   1:  PR[GP1:91,1] = PR[GP1:90,1] + -0.266;
   1:  PR[GP1:91,2] = PR[GP1:90,2] + -48.338;
   1:L PR[91] 10mm/sec CNT100;
   1:  PR[GP1:91,1] = PR[GP1:90,1] + 0.476;
   1:  PR[GP1:91,2] = PR[GP1:90,2] + -48.623;
   1:  PR[GP1:91,3] = PR[GP1:90,3] + 125.965;
   1:L PR[91] 10mm/sec CNT100;
   1:  PR[GP1:91,1] = PR[GP1:90,1] + 1.181;
   1:  PR[GP1:91,2] = PR[GP1:90,2] + -48.545;
   1:L PR[91] 10mm/sec CNT100;
   1:  PR[GP1:91,1] = PR[GP1:90,1] + 18.103;
   1:  PR[GP1:91,2] = PR[GP1:90,2] + -45.382;
   1:L PR[91] 10mm/sec CNT100;
   1:  PR[GP1:91,1] = PR[GP1:90,1] + 18.765;
   1:  PR[GP1:91,2] = PR[GP1:90,2] + -45.080;
   1:L PR[91] 10mm/sec CNT100;
   1:  PR[GP1:91,1] = PR[GP1:90,1] + 33.363;
   1:  PR[GP1:91,2] = PR[GP1:90,2] + -36.039;
   1:L PR[91] 10mm/sec CNT100;
   1:  PR[GP1:91,1] = PR[GP1:90,1] + 33.920;
   1:  PR[GP1:91,2] = PR[GP1:90,2] + -35.522;
   1:L PR[91] 10mm/sec CNT100;
   1:  PR[GP1:91,1] = PR[GP1:90,1] + 42.126;
   1:  PR[GP1:91,2] = PR[GP1:90,2] + -25.636;
   1:L PR[91] 10mm/sec CNT100;
   1:  PR[GP1:91,1] = PR[GP1:90,1] + 42.503;
   1:  PR[GP1:91,2] = PR[GP1:90,2] + -24.943;
   1:L PR[91] 10mm/sec CNT100;
   1:  PR[GP1:91,1] = PR[GP1:90,1] + 47.683;
   1:  PR[GP1:91,2] = PR[GP1:90,2] + -13.209;
   1:L PR[91] 10mm/sec CNT100;
   1:  PR[GP1:91,1] = PR[GP1:90,1] + 47.814;
   1:  PR[GP1:91,2] = PR[GP1:90,2] + -12.426;
   1:L PR[91] 10mm/sec CNT100;
   1:  PR[GP1:91,1] = PR[GP1:90,1] + 49.583;
   1:  PR[GP1:91,2] = PR[GP1:90,2] + 0.271;
   1:L PR[91] 10mm/sec CNT100;
   1:  PR[GP1:91,1] = PR[GP1:90,1] + 49.454;
   1:  PR[GP1:91,2] = PR[GP1:90,2] + 1.048;
   1:L PR[91] 10mm/sec CNT100;
   1:  PR[GP1:91,1] = PR[GP1:90,1] + 47.679;
   1:  PR[GP1:91,2] = PR[GP1:90,2] + 13.777;
   1:L PR[91] 10mm/sec CNT100;
   1:  PR[GP1:91,1] = PR[GP1:90,1] + 42.502;
   1:  PR[GP1:91,2] = PR[GP1:90,2] + 25.503;
   1:L PR[91] 10mm/sec CNT100;
   1:  PR[GP1:91,1] = PR[GP1:90,1] + 42.124;
   1:  PR[GP1:91,2] = PR[GP1:90,2] + 26.197;
   1:L PR[91] 10mm/sec CNT100;
   1:  PR[GP1:91,1] = PR[GP1:90,1] + 33.918;
   1:  PR[GP1:91,2] = PR[GP1:90,2] + 36.082;
   1:L PR[91] 10mm/sec CNT100;
   1:  PR[GP1:91,1] = PR[GP1:90,1] + 33.359;
   1:  PR[GP1:91,2] = PR[GP1:90,2] + 36.600;
   1:L PR[91] 10mm/sec CNT100;
   1:  PR[GP1:91,1] = PR[GP1:90,1] + 18.761;
   1:  PR[GP1:91,2] = PR[GP1:90,2] + 45.641;
   1:L PR[91] 10mm/sec CNT100;
   1:  PR[GP1:91,1] = PR[GP1:90,1] + 18.097;
   1:  PR[GP1:91,2] = PR[GP1:90,2] + 45.942;
   1:L PR[91] 10mm/sec CNT100;
   1:  PR[GP1:91,1] = PR[GP1:90,1] + 1.175;
   1:  PR[GP1:91,2] = PR[GP1:90,2] + 49.105;
   1:L PR[91] 10mm/sec CNT100;
   1:  PR[GP1:91,1] = PR[GP1:90,1] + 0.471;
   1:  PR[GP1:91,2] = PR[GP1:90,2] + 49.180;
   1:L PR[91] 10mm/sec CNT100;
   1:  PR[GP1:91,1] = PR[GP1:90,1] + -0.267;
   1:  PR[GP1:91,2] = PR[GP1:90,2] + 49.050;
   1:L PR[91] 10mm/sec CNT100;
   1:  PR[GP1:91,1] = PR[GP1:90,1] + -1.005;
   1:  PR[GP1:91,2] = PR[GP1:90,2] + 49.180;
   1:L PR[91] 10mm/sec CNT100;
   1:  PR[GP1:91,1] = PR[GP1:90,1] + -1.709;
   1:  PR[GP1:91,2] = PR[GP1:90,2] + 49.105;
   1:L PR[91] 10mm/sec CNT100;
   1:  PR[GP1:91,1] = PR[GP1:90,1] + -18.626;
   1:  PR[GP1:91,2] = PR[GP1:90,2] + 45.941;
   1:L PR[91] 10mm/sec CNT100;
   1:  PR[GP1:91,1] = PR[GP1:90,1] + -19.291;
   1:  PR[GP1:91,2] = PR[GP1:90,2] + 45.639;
   1:L PR[91] 10mm/sec CNT100;
   1:  PR[GP1:91,1] = PR[GP1:90,1] + -33.885;
   1:  PR[GP1:91,2] = PR[GP1:90,2] + 36.600;
   1:L PR[91] 10mm/sec CNT100;
   1:  PR[GP1:91,1] = PR[GP1:90,1] + -34.442;
   1:  PR[GP1:91,2] = PR[GP1:90,2] + 36.084;
   1:L PR[91] 10mm/sec CNT100;
   1:  PR[GP1:91,1] = PR[GP1:90,1] + -42.650;
   1:  PR[GP1:91,2] = PR[GP1:90,2] + 26.198;
   1:L PR[91] 10mm/sec CNT100;
   1:  PR[GP1:91,1] = PR[GP1:90,1] + -43.028;
   1:  PR[GP1:91,2] = PR[GP1:90,2] + 25.503;
   1:L PR[91] 10mm/sec CNT100;
   1:  PR[GP1:91,1] = PR[GP1:90,1] + -48.208;
   1:  PR[GP1:91,2] = PR[GP1:90,2] + 13.769;
   1:L PR[91] 10mm/sec CNT100;
   1:  PR[GP1:91,1] = PR[GP1:90,1] + -48.341;
   1:  PR[GP1:91,2] = PR[GP1:90,2] + 12.964;
   1:L PR[91] 10mm/sec CNT100;
   1:  PR[GP1:91,1] = PR[GP1:90,1] + -50.109;
   1:  PR[GP1:91,2] = PR[GP1:90,2] + 0.287;
   1:L PR[91] 10mm/sec CNT100;
   1:  PR[GP1:91,1] = PR[GP1:90,1] + -49.981;
   1:  PR[GP1:91,2] = PR[GP1:90,2] + -0.488;
   1:L PR[91] 10mm/sec CNT100;
   1:  PR[GP1:91,1] = PR[GP1:90,1] + -48.206;
   1:  PR[GP1:91,2] = PR[GP1:90,2] + -13.217;
   1:L PR[91] 10mm/sec CNT100;
   1:  PR[GP1:91,1] = PR[GP1:90,1] + -43.028;
   1:  PR[GP1:91,2] = PR[GP1:90,2] + -24.944;
   1:L PR[91] 10mm/sec CNT100;
   1:  PR[GP1:91,1] = PR[GP1:90,1] + -42.652;
   1:  PR[GP1:91,2] = PR[GP1:90,2] + -25.638;
   1:L PR[91] 10mm/sec CNT100;
   1:  PR[GP1:91,1] = PR[GP1:90,1] + -34.445;
   1:  PR[GP1:91,2] = PR[GP1:90,2] + -35.524;
   1:L PR[91] 10mm/sec CNT100;
   1:  PR[GP1:91,1] = PR[GP1:90,1] + -33.889;
   1:  PR[GP1:91,2] = PR[GP1:90,2] + -36.040;
   1:L PR[91] 10mm/sec CNT100;
   1:  PR[GP1:91,1] = PR[GP1:90,1] + -19.295;
   1:  PR[GP1:91,2] = PR[GP1:90,2] + -45.079;
   1:L PR[91] 10mm/sec CNT100;
   1:  PR[GP1:91,1] = PR[GP1:90,1] + -18.632;
   1:  PR[GP1:91,2] = PR[GP1:90,2] + -45.381;
   1:L PR[91] 10mm/sec CNT100;
   1:  PR[GP1:91,1] = PR[GP1:90,1] + -1.715;
   1:  PR[GP1:91,2] = PR[GP1:90,2] + -48.545;
   1:L PR[91] 10mm/sec CNT100;
   1:  PR[GP1:91,1] = PR[GP1:90,1] + -1.010;
   1:  PR[GP1:91,2] = PR[GP1:90,2] + -48.623;
   1:L PR[91] 10mm/sec CNT100;
   1:  PR[GP1:91,1] = PR[GP1:90,1] + -0.267;
   1:  PR[GP1:91,2] = PR[GP1:90,2] + -48.498;
   1:L PR[91] 10mm/sec CNT100;
   1:  PR[GP1:91,1] = PR[GP1:90,1] + 0.287;
   1:  PR[GP1:91,2] = PR[GP1:90,2] + -48.751;
   1:  PR[GP1:91,3] = PR[GP1:90,3] + 126.575;
   1:L PR[91] 10mm/sec CNT100;
   1:  PR[GP1:91,1] = PR[GP1:90,1] + 0.780;
   1:  PR[GP1:91,2] = PR[GP1:90,2] + -48.697;
   1:L PR[91] 10mm/sec CNT100;
   1:  PR[GP1:91,1] = PR[GP1:90,1] + 17.977;
   1:  PR[GP1:91,2] = PR[GP1:90,2] + -45.483;
   1:L PR[91] 10mm/sec CNT100;
   1:  PR[GP1:91,1] = PR[GP1:90,1] + 18.440;
   1:  PR[GP1:91,2] = PR[GP1:90,2] + -45.271;
   1:L PR[91] 10mm/sec CNT100;
   1:  PR[GP1:91,1] = PR[GP1:90,1] + 33.285;
   1:  PR[GP1:91,2] = PR[GP1:90,2] + -36.077;
   1:L PR[91] 10mm/sec CNT100;
   1:  PR[GP1:91,1] = PR[GP1:90,1] + 33.678;
   1:  PR[GP1:91,2] = PR[GP1:90,2] + -35.712;
   1:L PR[91] 10mm/sec CNT100;
   1:  PR[GP1:91,1] = PR[GP1:90,1] + 42.028;
   1:  PR[GP1:91,2] = PR[GP1:90,2] + -25.653;
   1:L PR[91] 10mm/sec CNT100;
   1:  PR[GP1:91,1] = PR[GP1:90,1] + 42.296;
   1:  PR[GP1:91,2] = PR[GP1:90,2] + -25.160;
   1:L PR[91] 10mm/sec CNT100;
   1:  PR[GP1:91,1] = PR[GP1:90,1] + 47.570;
   1:  PR[GP1:91,2] = PR[GP1:90,2] + -13.214;
   1:L PR[91] 10mm/sec CNT100;
   1:  PR[GP1:91,1] = PR[GP1:90,1] + 47.664;
   1:  PR[GP1:91,2] = PR[GP1:90,2] + -12.657;
   1:L PR[91] 10mm/sec CNT100;
   1:  PR[GP1:91,1] = PR[GP1:90,1] + 49.465;
   1:  PR[GP1:91,2] = PR[GP1:90,2] + 0.271;
   1:L PR[91] 10mm/sec CNT100;
   1:  PR[GP1:91,1] = PR[GP1:90,1] + 49.373;
   1:  PR[GP1:91,2] = PR[GP1:90,2] + 0.824;
   1:L PR[91] 10mm/sec CNT100;
   1:  PR[GP1:91,1] = PR[GP1:90,1] + 47.566;
   1:  PR[GP1:91,2] = PR[GP1:90,2] + 13.781;
   1:L PR[91] 10mm/sec CNT100;
   1:  PR[GP1:91,1] = PR[GP1:90,1] + 42.296;
   1:  PR[GP1:91,2] = PR[GP1:90,2] + 25.719;
   1:L PR[91] 10mm/sec CNT100;
   1:  PR[GP1:91,1] = PR[GP1:90,1] + 42.027;
   1:  PR[GP1:91,2] = PR[GP1:90,2] + 26.213;
   1:L PR[91] 10mm/sec CNT100;
   1:  PR[GP1:91,1] = PR[GP1:90,1] + 33.676;
   1:  PR[GP1:91,2] = PR[GP1:90,2] + 36.272;
   1:L PR[91] 10mm/sec CNT100;
   1:  PR[GP1:91,1] = PR[GP1:90,1] + 33.282;
   1:  PR[GP1:91,2] = PR[GP1:90,2] + 36.637;
   1:L PR[91] 10mm/sec CNT100;
   1:  PR[GP1:91,1] = PR[GP1:90,1] + 18.437;
   1:  PR[GP1:91,2] = PR[GP1:90,2] + 45.831;
   1:L PR[91] 10mm/sec CNT100;
   1:  PR[GP1:91,1] = PR[GP1:90,1] + 17.972;
   1:  PR[GP1:91,2] = PR[GP1:90,2] + 46.042;
   1:L PR[91] 10mm/sec CNT100;
   1:  PR[GP1:91,1] = PR[GP1:90,1] + 0.776;
   1:  PR[GP1:91,2] = PR[GP1:90,2] + 49.256;
   1:L PR[91] 10mm/sec CNT100;
   1:  PR[GP1:91,1] = PR[GP1:90,1] + 0.284;
   1:  PR[GP1:91,2] = PR[GP1:90,2] + 49.309;
   1:L PR[91] 10mm/sec CNT100;
   1:  PR[GP1:91,1] = PR[GP1:90,1] + -0.267;
   1:  PR[GP1:91,2] = PR[GP1:90,2] + 49.212;
   1:L PR[91] 10mm/sec CNT100;
   1:  PR[GP1:91,1] = PR[GP1:90,1] + -0.818;
   1:  PR[GP1:91,2] = PR[GP1:90,2] + 49.309;
   1:L PR[91] 10mm/sec CNT100;
   1:  PR[GP1:91,1] = PR[GP1:90,1] + -1.311;
   1:  PR[GP1:91,2] = PR[GP1:90,2] + 49.256;
   1:L PR[91] 10mm/sec CNT100;
   1:  PR[GP1:91,1] = PR[GP1:90,1] + -18.502;
   1:  PR[GP1:91,2] = PR[GP1:90,2] + 46.041;
   1:L PR[91] 10mm/sec CNT100;
   1:  PR[GP1:91,1] = PR[GP1:90,1] + -18.967;
   1:  PR[GP1:91,2] = PR[GP1:90,2] + 45.830;
   1:L PR[91] 10mm/sec CNT100;
   1:  PR[GP1:91,1] = PR[GP1:90,1] + -33.807;
   1:  PR[GP1:91,2] = PR[GP1:90,2] + 36.638;
   1:L PR[91] 10mm/sec CNT100;
   1:  PR[GP1:91,1] = PR[GP1:90,1] + -34.201;
   1:  PR[GP1:91,2] = PR[GP1:90,2] + 36.274;
   1:L PR[91] 10mm/sec CNT100;
   1:  PR[GP1:91,1] = PR[GP1:90,1] + -42.553;
   1:  PR[GP1:91,2] = PR[GP1:90,2] + 26.214;
   1:L PR[91] 10mm/sec CNT100;
   1:  PR[GP1:91,1] = PR[GP1:90,1] + -42.822;
   1:  PR[GP1:91,2] = PR[GP1:90,2] + 25.719;
   1:L PR[91] 10mm/sec CNT100;
   1:  PR[GP1:91,1] = PR[GP1:90,1] + -48.095;
   1:  PR[GP1:91,2] = PR[GP1:90,2] + 13.774;
   1:L PR[91] 10mm/sec CNT100;
   1:  PR[GP1:91,1] = PR[GP1:90,1] + -48.190;
   1:  PR[GP1:91,2] = PR[GP1:90,2] + 13.200;
   1:L PR[91] 10mm/sec CNT100;
   1:  PR[GP1:91,1] = PR[GP1:90,1] + -49.991;
   1:  PR[GP1:91,2] = PR[GP1:90,2] + 0.287;
   1:L PR[91] 10mm/sec CNT100;
   1:  PR[GP1:91,1] = PR[GP1:90,1] + -49.900;
   1:  PR[GP1:91,2] = PR[GP1:90,2] + -0.264;
   1:L PR[91] 10mm/sec CNT100;
   1:  PR[GP1:91,1] = PR[GP1:90,1] + -48.093;
   1:  PR[GP1:91,2] = PR[GP1:90,2] + -13.222;
   1:L PR[91] 10mm/sec CNT100;
   1:  PR[GP1:91,1] = PR[GP1:90,1] + -42.822;
   1:  PR[GP1:91,2] = PR[GP1:90,2] + -25.160;
   1:L PR[91] 10mm/sec CNT100;
   1:  PR[GP1:91,1] = PR[GP1:90,1] + -42.554;
   1:  PR[GP1:91,2] = PR[GP1:90,2] + -25.654;
   1:L PR[91] 10mm/sec CNT100;
   1:  PR[GP1:91,1] = PR[GP1:90,1] + -34.203;
   1:  PR[GP1:91,2] = PR[GP1:90,2] + -35.714;
   1:L PR[91] 10mm/sec CNT100;
   1:  PR[GP1:91,1] = PR[GP1:90,1] + -33.810;
   1:  PR[GP1:91,2] = PR[GP1:90,2] + -36.078;
   1:L PR[91] 10mm/sec CNT100;
   1:  PR[GP1:91,1] = PR[GP1:90,1] + -18.969;
   1:  PR[GP1:91,2] = PR[GP1:90,2] + -45.270;
   1:L PR[91] 10mm/sec CNT100;
   1:  PR[GP1:91,1] = PR[GP1:90,1] + -18.506;
   1:  PR[GP1:91,2] = PR[GP1:90,2] + -45.482;
   1:L PR[91] 10mm/sec CNT100;
   1:  PR[GP1:91,1] = PR[GP1:90,1] + -1.315;
   1:  PR[GP1:91,2] = PR[GP1:90,2] + -48.697;
   1:L PR[91] 10mm/sec CNT100;
   1:  PR[GP1:91,1] = PR[GP1:90,1] + -0.821;
   1:  PR[GP1:91,2] = PR[GP1:90,2] + -48.751;
   1:L PR[91] 10mm/sec CNT100;
   1:  PR[GP1:91,1] = PR[GP1:90,1] + -0.267;
   1:  PR[GP1:91,2] = PR[GP1:90,2] + -48.658;
   1:L PR[91] 10mm/sec CNT100;
   1:  PR[GP1:91,1] = PR[GP1:90,1] + 0.097;
   1:  PR[GP1:91,2] = PR[GP1:90,2] + -48.880;
   1:  PR[GP1:91,3] = PR[GP1:90,3] + 127.185;
   1:L PR[91] 10mm/sec CNT100;
   1:  PR[GP1:91,1] = PR[GP1:90,1] + 0.380;
   1:  PR[GP1:91,2] = PR[GP1:90,2] + -48.849;
   1:L PR[91] 10mm/sec CNT100;
   1:  PR[GP1:91,1] = PR[GP1:90,1] + 17.850;
   1:  PR[GP1:91,2] = PR[GP1:90,2] + -45.583;
   1:L PR[91] 10mm/sec CNT100;
   1:  PR[GP1:91,1] = PR[GP1:90,1] + 18.115;
   1:  PR[GP1:91,2] = PR[GP1:90,2] + -45.462;
   1:L PR[91] 10mm/sec CNT100;
   1:  PR[GP1:91,1] = PR[GP1:90,1] + 33.207;
   1:  PR[GP1:91,2] = PR[GP1:90,2] + -36.115;
   1:L PR[91] 10mm/sec CNT100;
   1:  PR[GP1:91,1] = PR[GP1:90,1] + 33.436;
   1:  PR[GP1:91,2] = PR[GP1:90,2] + -35.902;
   1:L PR[91] 10mm/sec CNT100;
   1:  PR[GP1:91,1] = PR[GP1:90,1] + 41.931;
   1:  PR[GP1:91,2] = PR[GP1:90,2] + -25.669;
   1:L PR[91] 10mm/sec CNT100;
   1:  PR[GP1:91,1] = PR[GP1:90,1] + 42.090;
   1:  PR[GP1:91,2] = PR[GP1:90,2] + -25.376;
   1:L PR[91] 10mm/sec CNT100;
   1:  PR[GP1:91,1] = PR[GP1:90,1] + 47.457;
   1:  PR[GP1:91,2] = PR[GP1:90,2] + -13.219;
   1:L PR[91] 10mm/sec CNT100;
   1:  PR[GP1:91,1] = PR[GP1:90,1] + 47.513;
   1:  PR[GP1:91,2] = PR[GP1:90,2] + -12.887;
   1:L PR[91] 10mm/sec CNT100;
   1:  PR[GP1:91,1] = PR[GP1:90,1] + 49.347;
   1:  PR[GP1:91,2] = PR[GP1:90,2] + 0.271;
   1:L PR[91] 10mm/sec CNT100;
   1:  PR[GP1:91,1] = PR[GP1:90,1] + 49.292;
   1:  PR[GP1:91,2] = PR[GP1:90,2] + 0.600;
   1:L PR[91] 10mm/sec CNT100;
   1:  PR[GP1:91,1] = PR[GP1:90,1] + 47.453;
   1:  PR[GP1:91,2] = PR[GP1:90,2] + 13.786;
   1:L PR[91] 10mm/sec CNT100;
   1:  PR[GP1:91,1] = PR[GP1:90,1] + 42.090;
   1:  PR[GP1:91,2] = PR[GP1:90,2] + 25.935;
   1:L PR[91] 10mm/sec CNT100;
   1:  PR[GP1:91,1] = PR[GP1:90,1] + 41.930;
   1:  PR[GP1:91,2] = PR[GP1:90,2] + 26.229;
   1:L PR[91] 10mm/sec CNT100;
   1:  PR[GP1:91,1] = PR[GP1:90,1] + 33.435;
   1:  PR[GP1:91,2] = PR[GP1:90,2] + 36.461;
   1:L PR[91] 10mm/sec CNT100;
   1:  PR[GP1:91,1] = PR[GP1:90,1] + 33.205;
   1:  PR[GP1:91,2] = PR[GP1:90,2] + 36.675;
   1:L PR[91] 10mm/sec CNT100;
   1:  PR[GP1:91,1] = PR[GP1:90,1] + 18.113;
   1:  PR[GP1:91,2] = PR[GP1:90,2] + 46.022;
   1:L PR[91] 10mm/sec CNT100;
   1:  PR[GP1:91,1] = PR[GP1:90,1] + 17.848;
   1:  PR[GP1:91,2] = PR[GP1:90,2] + 46.142;
   1:L PR[91] 10mm/sec CNT100;
   1:  PR[GP1:91,1] = PR[GP1:90,1] + 0.377;
   1:  PR[GP1:91,2] = PR[GP1:90,2] + 49.407;
   1:L PR[91] 10mm/sec CNT100;
   1:  PR[GP1:91,1] = PR[GP1:90,1] + 0.097;
   1:  PR[GP1:91,2] = PR[GP1:90,2] + 49.437;
   1:L PR[91] 10mm/sec CNT100;
   1:  PR[GP1:91,1] = PR[GP1:90,1] + -0.267;
   1:  PR[GP1:91,2] = PR[GP1:90,2] + 49.373;
   1:L PR[91] 10mm/sec CNT100;
   1:  PR[GP1:91,1] = PR[GP1:90,1] + -0.631;
   1:  PR[GP1:91,2] = PR[GP1:90,2] + 49.437;
   1:L PR[91] 10mm/sec CNT100;
   1:  PR[GP1:91,1] = PR[GP1:90,1] + -0.912;
   1:  PR[GP1:91,2] = PR[GP1:90,2] + 49.407;
   1:L PR[91] 10mm/sec CNT100;
   1:  PR[GP1:91,1] = PR[GP1:90,1] + -18.377;
   1:  PR[GP1:91,2] = PR[GP1:90,2] + 46.141;
   1:L PR[91] 10mm/sec CNT100;
   1:  PR[GP1:91,1] = PR[GP1:90,1] + -18.642;
   1:  PR[GP1:91,2] = PR[GP1:90,2] + 46.020;
   1:L PR[91] 10mm/sec CNT100;
   1:  PR[GP1:91,1] = PR[GP1:90,1] + -33.730;
   1:  PR[GP1:91,2] = PR[GP1:90,2] + 36.676;
   1:L PR[91] 10mm/sec CNT100;
   1:  PR[GP1:91,1] = PR[GP1:90,1] + -33.960;
   1:  PR[GP1:91,2] = PR[GP1:90,2] + 36.463;
   1:L PR[91] 10mm/sec CNT100;
   1:  PR[GP1:91,1] = PR[GP1:90,1] + -42.455;
   1:  PR[GP1:91,2] = PR[GP1:90,2] + 26.230;
   1:L PR[91] 10mm/sec CNT100;
   1:  PR[GP1:91,1] = PR[GP1:90,1] + -42.616;
   1:  PR[GP1:91,2] = PR[GP1:90,2] + 25.935;
   1:L PR[91] 10mm/sec CNT100;
   1:  PR[GP1:91,1] = PR[GP1:90,1] + -47.982;
   1:  PR[GP1:91,2] = PR[GP1:90,2] + 13.779;
   1:L PR[91] 10mm/sec CNT100;
   1:  PR[GP1:91,1] = PR[GP1:90,1] + -48.039;
   1:  PR[GP1:91,2] = PR[GP1:90,2] + 13.436;
   1:L PR[91] 10mm/sec CNT100;
   1:  PR[GP1:91,1] = PR[GP1:90,1] + -49.873;
   1:  PR[GP1:91,2] = PR[GP1:90,2] + 0.287;
   1:L PR[91] 10mm/sec CNT100;
   1:  PR[GP1:91,1] = PR[GP1:90,1] + -49.819;
   1:  PR[GP1:91,2] = PR[GP1:90,2] + -0.041;
   1:L PR[91] 10mm/sec CNT100;
   1:  PR[GP1:91,1] = PR[GP1:90,1] + -47.980;
   1:  PR[GP1:91,2] = PR[GP1:90,2] + -13.227;
   1:L PR[91] 10mm/sec CNT100;
   1:  PR[GP1:91,1] = PR[GP1:90,1] + -42.616;
   1:  PR[GP1:91,2] = PR[GP1:90,2] + -25.377;
   1:L PR[91] 10mm/sec CNT100;
   1:  PR[GP1:91,1] = PR[GP1:90,1] + -42.456;
   1:  PR[GP1:91,2] = PR[GP1:90,2] + -25.671;
   1:L PR[91] 10mm/sec CNT100;
   1:  PR[GP1:91,1] = PR[GP1:90,1] + -33.961;
   1:  PR[GP1:91,2] = PR[GP1:90,2] + -35.904;
   1:L PR[91] 10mm/sec CNT100;
   1:  PR[GP1:91,1] = PR[GP1:90,1] + -33.732;
   1:  PR[GP1:91,2] = PR[GP1:90,2] + -36.116;
   1:L PR[91] 10mm/sec CNT100;
   1:  PR[GP1:91,1] = PR[GP1:90,1] + -18.644;
   1:  PR[GP1:91,2] = PR[GP1:90,2] + -45.461;
   1:L PR[91] 10mm/sec CNT100;
   1:  PR[GP1:91,1] = PR[GP1:90,1] + -18.380;
   1:  PR[GP1:91,2] = PR[GP1:90,2] + -45.582;
   1:L PR[91] 10mm/sec CNT100;
   1:  PR[GP1:91,1] = PR[GP1:90,1] + -0.914;
   1:  PR[GP1:91,2] = PR[GP1:90,2] + -48.849;
   1:L PR[91] 10mm/sec CNT100;
   1:  PR[GP1:91,1] = PR[GP1:90,1] + -0.632;
   1:  PR[GP1:91,2] = PR[GP1:90,2] + -48.880;
   1:L PR[91] 10mm/sec CNT100;
   1:  PR[GP1:91,1] = PR[GP1:90,1] + -0.267;
   1:  PR[GP1:91,2] = PR[GP1:90,2] + -48.818;
   1:L PR[91] 10mm/sec CNT100;
   1:  PR[GP1:91,1] = PR[GP1:90,1] + -0.092;
   1:  PR[GP1:91,2] = PR[GP1:90,2] + -49.008;
   1:  PR[GP1:91,3] = PR[GP1:90,3] + 127.795;
   1:L PR[91] 10mm/sec CNT100;
   1:  PR[GP1:91,1] = PR[GP1:90,1] + -0.021;
   1:  PR[GP1:91,2] = PR[GP1:90,2] + -49.000;
   1:L PR[91] 10mm/sec CNT100;
   1:  PR[GP1:91,1] = PR[GP1:90,1] + 17.724;
   1:  PR[GP1:91,2] = PR[GP1:90,2] + -45.684;
   1:L PR[91] 10mm/sec CNT100;
   1:  PR[GP1:91,1] = PR[GP1:90,1] + 17.789;
   1:  PR[GP1:91,2] = PR[GP1:90,2] + -45.654;
   1:L PR[91] 10mm/sec CNT100;
   1:  PR[GP1:91,1] = PR[GP1:90,1] + 33.128;
   1:  PR[GP1:91,2] = PR[GP1:90,2] + -36.154;
   1:L PR[91] 10mm/sec CNT100;
   1:  PR[GP1:91,1] = PR[GP1:90,1] + 33.194;
   1:  PR[GP1:91,2] = PR[GP1:90,2] + -36.093;
   1:L PR[91] 10mm/sec CNT100;
   1:  PR[GP1:91,1] = PR[GP1:90,1] + 41.833;
   1:  PR[GP1:91,2] = PR[GP1:90,2] + -25.686;
   1:L PR[91] 10mm/sec CNT100;
   1:  PR[GP1:91,1] = PR[GP1:90,1] + 41.884;
   1:  PR[GP1:91,2] = PR[GP1:90,2] + -25.592;
   1:L PR[91] 10mm/sec CNT100;
   1:  PR[GP1:91,1] = PR[GP1:90,1] + 47.340;
   1:  PR[GP1:91,2] = PR[GP1:90,2] + -13.232;
   1:L PR[91] 10mm/sec CNT100;
   1:  PR[GP1:91,1] = PR[GP1:90,1] + 49.230;
   1:  PR[GP1:91,2] = PR[GP1:90,2] + 0.279;
   1:L PR[91] 10mm/sec CNT100;
   1:  PR[GP1:91,1] = PR[GP1:90,1] + 47.340;
   1:  PR[GP1:91,2] = PR[GP1:90,2] + 13.790;
   1:L PR[91] 10mm/sec CNT100;
   1:  PR[GP1:91,1] = PR[GP1:90,1] + 41.884;
   1:  PR[GP1:91,2] = PR[GP1:90,2] + 26.150;
   1:L PR[91] 10mm/sec CNT100;
   1:  PR[GP1:91,1] = PR[GP1:90,1] + 41.833;
   1:  PR[GP1:91,2] = PR[GP1:90,2] + 26.244;
   1:L PR[91] 10mm/sec CNT100;
   1:  PR[GP1:91,1] = PR[GP1:90,1] + 33.194;
   1:  PR[GP1:91,2] = PR[GP1:90,2] + 36.651;
   1:L PR[91] 10mm/sec CNT100;
   1:  PR[GP1:91,1] = PR[GP1:90,1] + 33.128;
   1:  PR[GP1:91,2] = PR[GP1:90,2] + 36.712;
   1:L PR[91] 10mm/sec CNT100;
   1:  PR[GP1:91,1] = PR[GP1:90,1] + 17.789;
   1:  PR[GP1:91,2] = PR[GP1:90,2] + 46.212;
   1:L PR[91] 10mm/sec CNT100;
   1:  PR[GP1:91,1] = PR[GP1:90,1] + 17.723;
   1:  PR[GP1:91,2] = PR[GP1:90,2] + 46.242;
   1:L PR[91] 10mm/sec CNT100;
   1:  PR[GP1:91,1] = PR[GP1:90,1] + -0.021;
   1:  PR[GP1:91,2] = PR[GP1:90,2] + 49.559;
   1:L PR[91] 10mm/sec CNT100;
   1:  PR[GP1:91,1] = PR[GP1:90,1] + -0.090;
   1:  PR[GP1:91,2] = PR[GP1:90,2] + 49.566;
   1:L PR[91] 10mm/sec CNT100;
   1:  PR[GP1:91,1] = PR[GP1:90,1] + -0.267;
   1:  PR[GP1:91,2] = PR[GP1:90,2] + 49.535;
   1:L PR[91] 10mm/sec CNT100;
   1:  PR[GP1:91,1] = PR[GP1:90,1] + -0.444;
   1:  PR[GP1:91,2] = PR[GP1:90,2] + 49.566;
   1:L PR[91] 10mm/sec CNT100;
   1:  PR[GP1:91,1] = PR[GP1:90,1] + -0.513;
   1:  PR[GP1:91,2] = PR[GP1:90,2] + 49.559;
   1:L PR[91] 10mm/sec CNT100;
   1:  PR[GP1:91,1] = PR[GP1:90,1] + -18.253;
   1:  PR[GP1:91,2] = PR[GP1:90,2] + 46.241;
   1:L PR[91] 10mm/sec CNT100;
   1:  PR[GP1:91,1] = PR[GP1:90,1] + -18.318;
   1:  PR[GP1:91,2] = PR[GP1:90,2] + 46.211;
   1:L PR[91] 10mm/sec CNT100;
   1:  PR[GP1:91,1] = PR[GP1:90,1] + -33.653;
   1:  PR[GP1:91,2] = PR[GP1:90,2] + 36.713;
   1:L PR[91] 10mm/sec CNT100;
   1:  PR[GP1:91,1] = PR[GP1:90,1] + -33.718;
   1:  PR[GP1:91,2] = PR[GP1:90,2] + 36.653;
   1:L PR[91] 10mm/sec CNT100;
   1:  PR[GP1:91,1] = PR[GP1:90,1] + -42.358;
   1:  PR[GP1:91,2] = PR[GP1:90,2] + 26.246;
   1:L PR[91] 10mm/sec CNT100;
   1:  PR[GP1:91,1] = PR[GP1:90,1] + -42.410;
   1:  PR[GP1:91,2] = PR[GP1:90,2] + 26.151;
   1:L PR[91] 10mm/sec CNT100;
   1:  PR[GP1:91,1] = PR[GP1:90,1] + -47.870;
   1:  PR[GP1:91,2] = PR[GP1:90,2] + 13.784;
   1:L PR[91] 10mm/sec CNT100;
   1:  PR[GP1:91,1] = PR[GP1:90,1] + -47.888;
   1:  PR[GP1:91,2] = PR[GP1:90,2] + 13.673;
   1:L PR[91] 10mm/sec CNT100;
   1:  PR[GP1:91,1] = PR[GP1:90,1] + -49.756;
   1:  PR[GP1:91,2] = PR[GP1:90,2] + 0.279;
   1:L PR[91] 10mm/sec CNT100;
   1:  PR[GP1:91,1] = PR[GP1:90,1] + -47.867;
   1:  PR[GP1:91,2] = PR[GP1:90,2] + -13.232;
   1:L PR[91] 10mm/sec CNT100;
   1:  PR[GP1:91,1] = PR[GP1:90,1] + -42.410;
   1:  PR[GP1:91,2] = PR[GP1:90,2] + -25.593;
   1:L PR[91] 10mm/sec CNT100;
   1:  PR[GP1:91,1] = PR[GP1:90,1] + -42.359;
   1:  PR[GP1:91,2] = PR[GP1:90,2] + -25.687;
   1:L PR[91] 10mm/sec CNT100;
   1:  PR[GP1:91,1] = PR[GP1:90,1] + -33.719;
   1:  PR[GP1:91,2] = PR[GP1:90,2] + -36.094;
   1:L PR[91] 10mm/sec CNT100;
   1:  PR[GP1:91,1] = PR[GP1:90,1] + -33.654;
   1:  PR[GP1:91,2] = PR[GP1:90,2] + -36.155;
   1:L PR[91] 10mm/sec CNT100;
   1:  PR[GP1:91,1] = PR[GP1:90,1] + -18.319;
   1:  PR[GP1:91,2] = PR[GP1:90,2] + -45.653;
   1:L PR[91] 10mm/sec CNT100;
   1:  PR[GP1:91,1] = PR[GP1:90,1] + -18.254;
   1:  PR[GP1:91,2] = PR[GP1:90,2] + -45.682;
   1:L PR[91] 10mm/sec CNT100;
   1:  PR[GP1:91,1] = PR[GP1:90,1] + -0.514;
   1:  PR[GP1:91,2] = PR[GP1:90,2] + -49.000;
   1:L PR[91] 10mm/sec CNT100;
   1:  PR[GP1:91,1] = PR[GP1:90,1] + -0.443;
   1:  PR[GP1:91,2] = PR[GP1:90,2] + -49.008;
   1:L PR[91] 10mm/sec CNT100;
   1:  PR[GP1:91,1] = PR[GP1:90,1] + -0.267;
   1:  PR[GP1:91,2] = PR[GP1:90,2] + -48.979;
   1:L PR[91] 10mm/sec CNT100;
   1:  PR[GP1:91,1] = PR[GP1:90,1] + 17.591;
   1:  PR[GP1:91,2] = PR[GP1:90,2] + -45.770;
   1:  PR[GP1:91,3] = PR[GP1:90,3] + 128.405;
   1:L PR[91] 10mm/sec CNT100;
   1:  PR[GP1:91,1] = PR[GP1:90,1] + 33.046;
   1:  PR[GP1:91,2] = PR[GP1:90,2] + -36.191;
   1:L PR[91] 10mm/sec CNT100;
   1:  PR[GP1:91,1] = PR[GP1:90,1] + 41.697;
   1:  PR[GP1:91,2] = PR[GP1:90,2] + -25.769;
   1:L PR[91] 10mm/sec CNT100;
   1:  PR[GP1:91,1] = PR[GP1:90,1] + 41.759;
   1:  PR[GP1:91,2] = PR[GP1:90,2] + -25.676;
   1:L PR[91] 10mm/sec CNT100;
   1:  PR[GP1:91,1] = PR[GP1:90,1] + 47.227;
   1:  PR[GP1:91,2] = PR[GP1:90,2] + -13.291;
   1:L PR[91] 10mm/sec CNT100;
   1:  PR[GP1:91,1] = PR[GP1:90,1] + 49.107;
   1:  PR[GP1:91,2] = PR[GP1:90,2] + 0.188;
   1:L PR[91] 10mm/sec CNT100;
   1:  PR[GP1:91,1] = PR[GP1:90,1] + 49.129;
   1:  PR[GP1:91,2] = PR[GP1:90,2] + 0.297;
   1:L PR[91] 10mm/sec CNT100;
   1:  PR[GP1:91,1] = PR[GP1:90,1] + 47.256;
   1:  PR[GP1:91,2] = PR[GP1:90,2] + 13.724;
   1:L PR[91] 10mm/sec CNT100;
   1:  PR[GP1:91,1] = PR[GP1:90,1] + 47.234;
   1:  PR[GP1:91,2] = PR[GP1:90,2] + 13.833;
   1:L PR[91] 10mm/sec CNT100;
   1:  PR[GP1:91,1] = PR[GP1:90,1] + 41.759;
   1:  PR[GP1:91,2] = PR[GP1:90,2] + 26.234;
   1:L PR[91] 10mm/sec CNT100;
   1:  PR[GP1:91,1] = PR[GP1:90,1] + 41.697;
   1:  PR[GP1:91,2] = PR[GP1:90,2] + 26.327;
   1:L PR[91] 10mm/sec CNT100;
   1:  PR[GP1:91,1] = PR[GP1:90,1] + 33.046;
   1:  PR[GP1:91,2] = PR[GP1:90,2] + 36.749;
   1:L PR[91] 10mm/sec CNT100;
   1:  PR[GP1:91,1] = PR[GP1:90,1] + 17.591;
   1:  PR[GP1:91,2] = PR[GP1:90,2] + 46.328;
   1:L PR[91] 10mm/sec CNT100;
   1:  PR[GP1:91,1] = PR[GP1:90,1] + -0.267;
   1:  PR[GP1:91,2] = PR[GP1:90,2] + 49.669;
   1:L PR[91] 10mm/sec CNT100;
   1:  PR[GP1:91,1] = PR[GP1:90,1] + -18.121;
   1:  PR[GP1:91,2] = PR[GP1:90,2] + 46.327;
   1:L PR[91] 10mm/sec CNT100;
   1:  PR[GP1:91,1] = PR[GP1:90,1] + -33.571;
   1:  PR[GP1:91,2] = PR[GP1:90,2] + 36.750;
   1:L PR[91] 10mm/sec CNT100;
   1:  PR[GP1:91,1] = PR[GP1:90,1] + -42.223;
   1:  PR[GP1:91,2] = PR[GP1:90,2] + 26.328;
   1:L PR[91] 10mm/sec CNT100;
   1:  PR[GP1:91,1] = PR[GP1:90,1] + -42.285;
   1:  PR[GP1:91,2] = PR[GP1:90,2] + 26.235;
   1:L PR[91] 10mm/sec CNT100;
   1:  PR[GP1:91,1] = PR[GP1:90,1] + -47.753;
   1:  PR[GP1:91,2] = PR[GP1:90,2] + 13.849;
   1:L PR[91] 10mm/sec CNT100;
   1:  PR[GP1:91,1] = PR[GP1:90,1] + -49.633;
   1:  PR[GP1:91,2] = PR[GP1:90,2] + 0.370;
   1:L PR[91] 10mm/sec CNT100;
   1:  PR[GP1:91,1] = PR[GP1:90,1] + -49.655;
   1:  PR[GP1:91,2] = PR[GP1:90,2] + 0.261;
   1:L PR[91] 10mm/sec CNT100;
   1:  PR[GP1:91,1] = PR[GP1:90,1] + -47.782;
   1:  PR[GP1:91,2] = PR[GP1:90,2] + -13.166;
   1:L PR[91] 10mm/sec CNT100;
   1:  PR[GP1:91,1] = PR[GP1:90,1] + -47.760;
   1:  PR[GP1:91,2] = PR[GP1:90,2] + -13.275;
   1:L PR[91] 10mm/sec CNT100;
   1:  PR[GP1:91,1] = PR[GP1:90,1] + -42.285;
   1:  PR[GP1:91,2] = PR[GP1:90,2] + -25.677;
   1:L PR[91] 10mm/sec CNT100;
   1:  PR[GP1:91,1] = PR[GP1:90,1] + -42.223;
   1:  PR[GP1:91,2] = PR[GP1:90,2] + -25.770;
   1:L PR[91] 10mm/sec CNT100;
   1:  PR[GP1:91,1] = PR[GP1:90,1] + -33.571;
   1:  PR[GP1:91,2] = PR[GP1:90,2] + -36.191;
   1:L PR[91] 10mm/sec CNT100;
   1:  PR[GP1:91,1] = PR[GP1:90,1] + -18.121;
   1:  PR[GP1:91,2] = PR[GP1:90,2] + -45.769;
   1:L PR[91] 10mm/sec CNT100;
   1:  PR[GP1:91,1] = PR[GP1:90,1] + -0.267;
   1:  PR[GP1:91,2] = PR[GP1:90,2] + -49.111;
   1:L PR[91] 10mm/sec CNT100;
   1:  PR[GP1:91,1] = PR[GP1:90,1] + 16.405;
   1:  PR[GP1:91,2] = PR[GP1:90,2] + -45.994;
   1:  PR[GP1:91,3] = PR[GP1:90,3] + 129.015;
   1:L PR[91] 10mm/sec CNT100;
   1:  PR[GP1:91,1] = PR[GP1:90,1] + 17.653;
   1:  PR[GP1:91,2] = PR[GP1:90,2] + -45.746;
   1:L PR[91] 10mm/sec CNT100;
   1:  PR[GP1:91,1] = PR[GP1:90,1] + 32.071;
   1:  PR[GP1:91,2] = PR[GP1:90,2] + -36.817;
   1:L PR[91] 10mm/sec CNT100;
   1:  PR[GP1:91,1] = PR[GP1:90,1] + 33.141;
   1:  PR[GP1:91,2] = PR[GP1:90,2] + -36.102;
   1:L PR[91] 10mm/sec CNT100;
   1:  PR[GP1:91,1] = PR[GP1:90,1] + 41.261;
   1:  PR[GP1:91,2] = PR[GP1:90,2] + -26.320;
   1:L PR[91] 10mm/sec CNT100;
   1:  PR[GP1:91,1] = PR[GP1:90,1] + 41.984;
   1:  PR[GP1:91,2] = PR[GP1:90,2] + -25.238;
   1:L PR[91] 10mm/sec CNT100;
   1:  PR[GP1:91,1] = PR[GP1:90,1] + 47.111;
   1:  PR[GP1:91,2] = PR[GP1:90,2] + -13.623;
   1:L PR[91] 10mm/sec CNT100;
   1:  PR[GP1:91,1] = PR[GP1:90,1] + 48.875;
   1:  PR[GP1:91,2] = PR[GP1:90,2] + -0.979;
   1:L PR[91] 10mm/sec CNT100;
   1:  PR[GP1:91,1] = PR[GP1:90,1] + 49.129;
   1:  PR[GP1:91,2] = PR[GP1:90,2] + 0.297;
   1:L PR[91] 10mm/sec CNT100;
   1:  PR[GP1:91,1] = PR[GP1:90,1] + 47.372;
   1:  PR[GP1:91,2] = PR[GP1:90,2] + 12.889;
   1:L PR[91] 10mm/sec CNT100;
   1:  PR[GP1:91,1] = PR[GP1:90,1] + 47.118;
   1:  PR[GP1:91,2] = PR[GP1:90,2] + 14.165;
   1:L PR[91] 10mm/sec CNT100;
   1:  PR[GP1:91,1] = PR[GP1:90,1] + 41.984;
   1:  PR[GP1:91,2] = PR[GP1:90,2] + 25.796;
   1:L PR[91] 10mm/sec CNT100;
   1:  PR[GP1:91,1] = PR[GP1:90,1] + 41.261;
   1:  PR[GP1:91,2] = PR[GP1:90,2] + 26.878;
   1:L PR[91] 10mm/sec CNT100;
   1:  PR[GP1:91,1] = PR[GP1:90,1] + 33.141;
   1:  PR[GP1:91,2] = PR[GP1:90,2] + 36.660;
   1:L PR[91] 10mm/sec CNT100;
   1:  PR[GP1:91,1] = PR[GP1:90,1] + 32.071;
   1:  PR[GP1:91,2] = PR[GP1:90,2] + 37.375;
   1:L PR[91] 10mm/sec CNT100;
   1:  PR[GP1:91,1] = PR[GP1:90,1] + 17.653;
   1:  PR[GP1:91,2] = PR[GP1:90,2] + 46.304;
   1:L PR[91] 10mm/sec CNT100;
   1:  PR[GP1:91,1] = PR[GP1:90,1] + 16.405;
   1:  PR[GP1:91,2] = PR[GP1:90,2] + 46.552;
   1:L PR[91] 10mm/sec CNT100;
   1:  PR[GP1:91,1] = PR[GP1:90,1] + -0.267;
   1:  PR[GP1:91,2] = PR[GP1:90,2] + 49.669;
   1:L PR[91] 10mm/sec CNT100;
   1:  PR[GP1:91,1] = PR[GP1:90,1] + -16.934;
   1:  PR[GP1:91,2] = PR[GP1:90,2] + 46.551;
   1:L PR[91] 10mm/sec CNT100;
   1:  PR[GP1:91,1] = PR[GP1:90,1] + -18.183;
   1:  PR[GP1:91,2] = PR[GP1:90,2] + 46.303;
   1:L PR[91] 10mm/sec CNT100;
   1:  PR[GP1:91,1] = PR[GP1:90,1] + -32.594;
   1:  PR[GP1:91,2] = PR[GP1:90,2] + 37.377;
   1:L PR[91] 10mm/sec CNT100;
   1:  PR[GP1:91,1] = PR[GP1:90,1] + -33.666;
   1:  PR[GP1:91,2] = PR[GP1:90,2] + 36.661;
   1:L PR[91] 10mm/sec CNT100;
   1:  PR[GP1:91,1] = PR[GP1:90,1] + -41.787;
   1:  PR[GP1:91,2] = PR[GP1:90,2] + 26.879;
   1:L PR[91] 10mm/sec CNT100;
   1:  PR[GP1:91,1] = PR[GP1:90,1] + -42.510;
   1:  PR[GP1:91,2] = PR[GP1:90,2] + 25.797;
   1:L PR[91] 10mm/sec CNT100;
   1:  PR[GP1:91,1] = PR[GP1:90,1] + -47.637;
   1:  PR[GP1:91,2] = PR[GP1:90,2] + 14.182;
   1:L PR[91] 10mm/sec CNT100;
   1:  PR[GP1:91,1] = PR[GP1:90,1] + -49.401;
   1:  PR[GP1:91,2] = PR[GP1:90,2] + 1.537;
   1:L PR[91] 10mm/sec CNT100;
   1:  PR[GP1:91,1] = PR[GP1:90,1] + -49.655;
   1:  PR[GP1:91,2] = PR[GP1:90,2] + 0.261;
   1:L PR[91] 10mm/sec CNT100;
   1:  PR[GP1:91,1] = PR[GP1:90,1] + -47.898;
   1:  PR[GP1:91,2] = PR[GP1:90,2] + -12.331;
   1:L PR[91] 10mm/sec CNT100;
   1:  PR[GP1:91,1] = PR[GP1:90,1] + -47.645;
   1:  PR[GP1:91,2] = PR[GP1:90,2] + -13.608;
   1:L PR[91] 10mm/sec CNT100;
   1:  PR[GP1:91,1] = PR[GP1:90,1] + -42.510;
   1:  PR[GP1:91,2] = PR[GP1:90,2] + -25.239;
   1:L PR[91] 10mm/sec CNT100;
   1:  PR[GP1:91,1] = PR[GP1:90,1] + -41.787;
   1:  PR[GP1:91,2] = PR[GP1:90,2] + -26.321;
   1:L PR[91] 10mm/sec CNT100;
   1:  PR[GP1:91,1] = PR[GP1:90,1] + -33.666;
   1:  PR[GP1:91,2] = PR[GP1:90,2] + -36.103;
   1:L PR[91] 10mm/sec CNT100;
   1:  PR[GP1:91,1] = PR[GP1:90,1] + -32.594;
   1:  PR[GP1:91,2] = PR[GP1:90,2] + -36.819;
   1:L PR[91] 10mm/sec CNT100;
   1:  PR[GP1:91,1] = PR[GP1:90,1] + -18.186;
   1:  PR[GP1:91,2] = PR[GP1:90,2] + -45.743;
   1:L PR[91] 10mm/sec CNT100;
   1:  PR[GP1:91,1] = PR[GP1:90,1] + -1.512;
   1:  PR[GP1:91,2] = PR[GP1:90,2] + -48.862;
   1:L PR[91] 10mm/sec CNT100;
   1:  PR[GP1:91,1] = PR[GP1:90,1] + -0.264;
   1:  PR[GP1:91,2] = PR[GP1:90,2] + -49.110;
   1:L PR[91] 10mm/sec CNT100;
   1:  PR[GP1:91,1] = PR[GP1:90,1] + 15.303;
   1:  PR[GP1:91,2] = PR[GP1:90,2] + -46.200;
   1:  PR[GP1:91,3] = PR[GP1:90,3] + 129.625;
   1:L PR[91] 10mm/sec CNT100;
   1:  PR[GP1:91,1] = PR[GP1:90,1] + 17.719;
   1:  PR[GP1:91,2] = PR[GP1:90,2] + -45.720;
   1:L PR[91] 10mm/sec CNT100;
   1:  PR[GP1:91,1] = PR[GP1:90,1] + 31.183;
   1:  PR[GP1:91,2] = PR[GP1:90,2] + -37.381;
   1:L PR[91] 10mm/sec CNT100;
   1:  PR[GP1:91,1] = PR[GP1:90,1] + 33.242;
   1:  PR[GP1:91,2] = PR[GP1:90,2] + -36.005;
   1:L PR[91] 10mm/sec CNT100;
   1:  PR[GP1:91,1] = PR[GP1:90,1] + 40.824;
   1:  PR[GP1:91,2] = PR[GP1:90,2] + -26.872;
   1:L PR[91] 10mm/sec CNT100;
   1:  PR[GP1:91,1] = PR[GP1:90,1] + 42.208;
   1:  PR[GP1:91,2] = PR[GP1:90,2] + -24.800;
   1:L PR[91] 10mm/sec CNT100;
   1:  PR[GP1:91,1] = PR[GP1:90,1] + 46.995;
   1:  PR[GP1:91,2] = PR[GP1:90,2] + -13.956;
   1:L PR[91] 10mm/sec CNT100;
   1:  PR[GP1:91,1] = PR[GP1:90,1] + 48.643;
   1:  PR[GP1:91,2] = PR[GP1:90,2] + -2.146;
   1:L PR[91] 10mm/sec CNT100;
   1:  PR[GP1:91,1] = PR[GP1:90,1] + 49.129;
   1:  PR[GP1:91,2] = PR[GP1:90,2] + 0.297;
   1:L PR[91] 10mm/sec CNT100;
   1:  PR[GP1:91,1] = PR[GP1:90,1] + 47.489;
   1:  PR[GP1:91,2] = PR[GP1:90,2] + 12.054;
   1:L PR[91] 10mm/sec CNT100;
   1:  PR[GP1:91,1] = PR[GP1:90,1] + 47.002;
   1:  PR[GP1:91,2] = PR[GP1:90,2] + 14.498;
   1:L PR[91] 10mm/sec CNT100;
   1:  PR[GP1:91,1] = PR[GP1:90,1] + 42.208;
   1:  PR[GP1:91,2] = PR[GP1:90,2] + 25.358;
   1:L PR[91] 10mm/sec CNT100;
   1:  PR[GP1:91,1] = PR[GP1:90,1] + 40.824;
   1:  PR[GP1:91,2] = PR[GP1:90,2] + 27.430;
   1:L PR[91] 10mm/sec CNT100;
   1:  PR[GP1:91,1] = PR[GP1:90,1] + 33.242;
   1:  PR[GP1:91,2] = PR[GP1:90,2] + 36.563;
   1:L PR[91] 10mm/sec CNT100;
   1:  PR[GP1:91,1] = PR[GP1:90,1] + 31.183;
   1:  PR[GP1:91,2] = PR[GP1:90,2] + 37.939;
   1:L PR[91] 10mm/sec CNT100;
   1:  PR[GP1:91,1] = PR[GP1:90,1] + 17.719;
   1:  PR[GP1:91,2] = PR[GP1:90,2] + 46.278;
   1:L PR[91] 10mm/sec CNT100;
   1:  PR[GP1:91,1] = PR[GP1:90,1] + 15.303;
   1:  PR[GP1:91,2] = PR[GP1:90,2] + 46.758;
   1:L PR[91] 10mm/sec CNT100;
   1:  PR[GP1:91,1] = PR[GP1:90,1] + -0.267;
   1:  PR[GP1:91,2] = PR[GP1:90,2] + 49.669;
   1:L PR[91] 10mm/sec CNT100;
   1:  PR[GP1:91,1] = PR[GP1:90,1] + -15.831;
   1:  PR[GP1:91,2] = PR[GP1:90,2] + 46.757;
   1:L PR[91] 10mm/sec CNT100;
   1:  PR[GP1:91,1] = PR[GP1:90,1] + -18.248;
   1:  PR[GP1:91,2] = PR[GP1:90,2] + 46.277;
   1:L PR[91] 10mm/sec CNT100;
   1:  PR[GP1:91,1] = PR[GP1:90,1] + -31.706;
   1:  PR[GP1:91,2] = PR[GP1:90,2] + 37.941;
   1:L PR[91] 10mm/sec CNT100;
   1:  PR[GP1:91,1] = PR[GP1:90,1] + -33.768;
   1:  PR[GP1:91,2] = PR[GP1:90,2] + 36.564;
   1:L PR[91] 10mm/sec CNT100;
   1:  PR[GP1:91,1] = PR[GP1:90,1] + -41.350;
   1:  PR[GP1:91,2] = PR[GP1:90,2] + 27.431;
   1:L PR[91] 10mm/sec CNT100;
   1:  PR[GP1:91,1] = PR[GP1:90,1] + -42.734;
   1:  PR[GP1:91,2] = PR[GP1:90,2] + 25.359;
   1:L PR[91] 10mm/sec CNT100;
   1:  PR[GP1:91,1] = PR[GP1:90,1] + -47.522;
   1:  PR[GP1:91,2] = PR[GP1:90,2] + 14.514;
   1:L PR[91] 10mm/sec CNT100;
   1:  PR[GP1:91,1] = PR[GP1:90,1] + -49.169;
   1:  PR[GP1:91,2] = PR[GP1:90,2] + 2.704;
   1:L PR[91] 10mm/sec CNT100;
   1:  PR[GP1:91,1] = PR[GP1:90,1] + -49.655;
   1:  PR[GP1:91,2] = PR[GP1:90,2] + 0.261;
   1:L PR[91] 10mm/sec CNT100;
   1:  PR[GP1:91,1] = PR[GP1:90,1] + -48.015;
   1:  PR[GP1:91,2] = PR[GP1:90,2] + -11.497;
   1:L PR[91] 10mm/sec CNT100;
   1:  PR[GP1:91,1] = PR[GP1:90,1] + -47.529;
   1:  PR[GP1:91,2] = PR[GP1:90,2] + -13.940;
   1:L PR[91] 10mm/sec CNT100;
   1:  PR[GP1:91,1] = PR[GP1:90,1] + -42.734;
   1:  PR[GP1:91,2] = PR[GP1:90,2] + -24.801;
   1:L PR[91] 10mm/sec CNT100;
   1:  PR[GP1:91,1] = PR[GP1:90,1] + -41.350;
   1:  PR[GP1:91,2] = PR[GP1:90,2] + -26.872;
   1:L PR[91] 10mm/sec CNT100;
   1:  PR[GP1:91,1] = PR[GP1:90,1] + -33.768;
   1:  PR[GP1:91,2] = PR[GP1:90,2] + -36.006;
   1:L PR[91] 10mm/sec CNT100;
   1:  PR[GP1:91,1] = PR[GP1:90,1] + -31.706;
   1:  PR[GP1:91,2] = PR[GP1:90,2] + -37.383;
   1:L PR[91] 10mm/sec CNT100;
   1:  PR[GP1:91,1] = PR[GP1:90,1] + -18.251;
   1:  PR[GP1:91,2] = PR[GP1:90,2] + -45.717;
   1:L PR[91] 10mm/sec CNT100;
   1:  PR[GP1:91,1] = PR[GP1:90,1] + -2.679;
   1:  PR[GP1:91,2] = PR[GP1:90,2] + -48.629;
   1:L PR[91] 10mm/sec CNT100;
   1:  PR[GP1:91,1] = PR[GP1:90,1] + -0.263;
   1:  PR[GP1:91,2] = PR[GP1:90,2] + -49.110;
   1:L PR[91] 10mm/sec CNT100;
   1:  PR[GP1:91,1] = PR[GP1:90,1] + 14.201;
   1:  PR[GP1:91,2] = PR[GP1:90,2] + -46.406;
   1:  PR[GP1:91,3] = PR[GP1:90,3] + 130.235;
   1:L PR[91] 10mm/sec CNT100;
   1:  PR[GP1:91,1] = PR[GP1:90,1] + 17.784;
   1:  PR[GP1:91,2] = PR[GP1:90,2] + -45.694;
   1:L PR[91] 10mm/sec CNT100;
   1:  PR[GP1:91,1] = PR[GP1:90,1] + 30.295;
   1:  PR[GP1:91,2] = PR[GP1:90,2] + -37.945;
   1:L PR[91] 10mm/sec CNT100;
   1:  PR[GP1:91,1] = PR[GP1:90,1] + 33.344;
   1:  PR[GP1:91,2] = PR[GP1:90,2] + -35.908;
   1:L PR[91] 10mm/sec CNT100;
   1:  PR[GP1:91,1] = PR[GP1:90,1] + 40.387;
   1:  PR[GP1:91,2] = PR[GP1:90,2] + -27.423;
   1:L PR[91] 10mm/sec CNT100;
   1:  PR[GP1:91,1] = PR[GP1:90,1] + 42.433;
   1:  PR[GP1:91,2] = PR[GP1:90,2] + -24.362;
   1:L PR[91] 10mm/sec CNT100;
   1:  PR[GP1:91,1] = PR[GP1:90,1] + 46.880;
   1:  PR[GP1:91,2] = PR[GP1:90,2] + -14.289;
   1:L PR[91] 10mm/sec CNT100;
   1:  PR[GP1:91,1] = PR[GP1:90,1] + 48.410;
   1:  PR[GP1:91,2] = PR[GP1:90,2] + -3.313;
   1:L PR[91] 10mm/sec CNT100;
   1:  PR[GP1:91,1] = PR[GP1:90,1] + 49.129;
   1:  PR[GP1:91,2] = PR[GP1:90,2] + 0.297;
   1:L PR[91] 10mm/sec CNT100;
   1:  PR[GP1:91,1] = PR[GP1:90,1] + 47.605;
   1:  PR[GP1:91,2] = PR[GP1:90,2] + 11.220;
   1:L PR[91] 10mm/sec CNT100;
   1:  PR[GP1:91,1] = PR[GP1:90,1] + 46.887;
   1:  PR[GP1:91,2] = PR[GP1:90,2] + 14.831;
   1:L PR[91] 10mm/sec CNT100;
   1:  PR[GP1:91,1] = PR[GP1:90,1] + 42.433;
   1:  PR[GP1:91,2] = PR[GP1:90,2] + 24.920;
   1:L PR[91] 10mm/sec CNT100;
   1:  PR[GP1:91,1] = PR[GP1:90,1] + 40.387;
   1:  PR[GP1:91,2] = PR[GP1:90,2] + 27.981;
   1:L PR[91] 10mm/sec CNT100;
   1:  PR[GP1:91,1] = PR[GP1:90,1] + 33.344;
   1:  PR[GP1:91,2] = PR[GP1:90,2] + 36.466;
   1:L PR[91] 10mm/sec CNT100;
   1:  PR[GP1:91,1] = PR[GP1:90,1] + 30.295;
   1:  PR[GP1:91,2] = PR[GP1:90,2] + 38.503;
   1:L PR[91] 10mm/sec CNT100;
   1:  PR[GP1:91,1] = PR[GP1:90,1] + 17.784;
   1:  PR[GP1:91,2] = PR[GP1:90,2] + 46.252;
   1:L PR[91] 10mm/sec CNT100;
   1:  PR[GP1:91,1] = PR[GP1:90,1] + 14.201;
   1:  PR[GP1:91,2] = PR[GP1:90,2] + 46.964;
   1:L PR[91] 10mm/sec CNT100;
   1:  PR[GP1:91,1] = PR[GP1:90,1] + -0.267;
   1:  PR[GP1:91,2] = PR[GP1:90,2] + 49.669;
   1:L PR[91] 10mm/sec CNT100;
   1:  PR[GP1:91,1] = PR[GP1:90,1] + -14.729;
   1:  PR[GP1:91,2] = PR[GP1:90,2] + 46.964;
   1:L PR[91] 10mm/sec CNT100;
   1:  PR[GP1:91,1] = PR[GP1:90,1] + -18.313;
   1:  PR[GP1:91,2] = PR[GP1:90,2] + 46.251;
   1:L PR[91] 10mm/sec CNT100;
   1:  PR[GP1:91,1] = PR[GP1:90,1] + -30.818;
   1:  PR[GP1:91,2] = PR[GP1:90,2] + 38.505;
   1:L PR[91] 10mm/sec CNT100;
   1:  PR[GP1:91,1] = PR[GP1:90,1] + -33.869;
   1:  PR[GP1:91,2] = PR[GP1:90,2] + 36.467;
   1:L PR[91] 10mm/sec CNT100;
   1:  PR[GP1:91,1] = PR[GP1:90,1] + -40.913;
   1:  PR[GP1:91,2] = PR[GP1:90,2] + 27.982;
   1:L PR[91] 10mm/sec CNT100;
   1:  PR[GP1:91,1] = PR[GP1:90,1] + -42.959;
   1:  PR[GP1:91,2] = PR[GP1:90,2] + 24.920;
   1:L PR[91] 10mm/sec CNT100;
   1:  PR[GP1:91,1] = PR[GP1:90,1] + -47.406;
   1:  PR[GP1:91,2] = PR[GP1:90,2] + 14.847;
   1:L PR[91] 10mm/sec CNT100;
   1:  PR[GP1:91,1] = PR[GP1:90,1] + -48.937;
   1:  PR[GP1:91,2] = PR[GP1:90,2] + 3.871;
   1:L PR[91] 10mm/sec CNT100;
   1:  PR[GP1:91,1] = PR[GP1:90,1] + -49.655;
   1:  PR[GP1:91,2] = PR[GP1:90,2] + 0.261;
   1:L PR[91] 10mm/sec CNT100;
   1:  PR[GP1:91,1] = PR[GP1:90,1] + -48.131;
   1:  PR[GP1:91,2] = PR[GP1:90,2] + -10.662;
   1:L PR[91] 10mm/sec CNT100;
   1:  PR[GP1:91,1] = PR[GP1:90,1] + -47.413;
   1:  PR[GP1:91,2] = PR[GP1:90,2] + -14.273;
   1:L PR[91] 10mm/sec CNT100;
   1:  PR[GP1:91,1] = PR[GP1:90,1] + -42.959;
   1:  PR[GP1:91,2] = PR[GP1:90,2] + -24.362;
   1:L PR[91] 10mm/sec CNT100;
   1:  PR[GP1:91,1] = PR[GP1:90,1] + -40.913;
   1:  PR[GP1:91,2] = PR[GP1:90,2] + -27.424;
   1:L PR[91] 10mm/sec CNT100;
   1:  PR[GP1:91,1] = PR[GP1:90,1] + -33.869;
   1:  PR[GP1:91,2] = PR[GP1:90,2] + -35.909;
   1:L PR[91] 10mm/sec CNT100;
   1:  PR[GP1:91,1] = PR[GP1:90,1] + -30.818;
   1:  PR[GP1:91,2] = PR[GP1:90,2] + -37.947;
   1:L PR[91] 10mm/sec CNT100;
   1:  PR[GP1:91,1] = PR[GP1:90,1] + -18.316;
   1:  PR[GP1:91,2] = PR[GP1:90,2] + -45.691;
   1:L PR[91] 10mm/sec CNT100;
   1:  PR[GP1:91,1] = PR[GP1:90,1] + -3.846;
   1:  PR[GP1:91,2] = PR[GP1:90,2] + -48.397;
   1:L PR[91] 10mm/sec CNT100;
   1:  PR[GP1:91,1] = PR[GP1:90,1] + -0.263;
   1:  PR[GP1:91,2] = PR[GP1:90,2] + -49.110;
   1:L PR[91] 10mm/sec CNT100;
   1:  PR[GP1:91,1] = PR[GP1:90,1] + 13.099;
   1:  PR[GP1:91,2] = PR[GP1:90,2] + -46.612;
   1:  PR[GP1:91,3] = PR[GP1:90,3] + 130.845;
   1:L PR[91] 10mm/sec CNT100;
   1:  PR[GP1:91,1] = PR[GP1:90,1] + 17.849;
   1:  PR[GP1:91,2] = PR[GP1:90,2] + -45.667;
   1:L PR[91] 10mm/sec CNT100;
   1:  PR[GP1:91,1] = PR[GP1:90,1] + 29.407;
   1:  PR[GP1:91,2] = PR[GP1:90,2] + -38.509;
   1:L PR[91] 10mm/sec CNT100;
   1:  PR[GP1:91,1] = PR[GP1:90,1] + 33.445;
   1:  PR[GP1:91,2] = PR[GP1:90,2] + -35.811;
   1:L PR[91] 10mm/sec CNT100;
   1:  PR[GP1:91,1] = PR[GP1:90,1] + 39.951;
   1:  PR[GP1:91,2] = PR[GP1:90,2] + -27.974;
   1:L PR[91] 10mm/sec CNT100;
   1:  PR[GP1:91,1] = PR[GP1:90,1] + 42.657;
   1:  PR[GP1:91,2] = PR[GP1:90,2] + -23.924;
   1:L PR[91] 10mm/sec CNT100;
   1:  PR[GP1:91,1] = PR[GP1:90,1] + 46.764;
   1:  PR[GP1:91,2] = PR[GP1:90,2] + -14.621;
   1:L PR[91] 10mm/sec CNT100;
   1:  PR[GP1:91,1] = PR[GP1:90,1] + 48.178;
   1:  PR[GP1:91,2] = PR[GP1:90,2] + -4.481;
   1:L PR[91] 10mm/sec CNT100;
   1:  PR[GP1:91,1] = PR[GP1:90,1] + 49.129;
   1:  PR[GP1:91,2] = PR[GP1:90,2] + 0.297;
   1:L PR[91] 10mm/sec CNT100;
   1:  PR[GP1:91,1] = PR[GP1:90,1] + 47.721;
   1:  PR[GP1:91,2] = PR[GP1:90,2] + 10.385;
   1:L PR[91] 10mm/sec CNT100;
   1:  PR[GP1:91,1] = PR[GP1:90,1] + 46.771;
   1:  PR[GP1:91,2] = PR[GP1:90,2] + 15.163;
   1:L PR[91] 10mm/sec CNT100;
   1:  PR[GP1:91,1] = PR[GP1:90,1] + 42.657;
   1:  PR[GP1:91,2] = PR[GP1:90,2] + 24.482;
   1:L PR[91] 10mm/sec CNT100;
   1:  PR[GP1:91,1] = PR[GP1:90,1] + 39.951;
   1:  PR[GP1:91,2] = PR[GP1:90,2] + 28.532;
   1:L PR[91] 10mm/sec CNT100;
   1:  PR[GP1:91,1] = PR[GP1:90,1] + 33.445;
   1:  PR[GP1:91,2] = PR[GP1:90,2] + 36.369;
   1:L PR[91] 10mm/sec CNT100;
   1:  PR[GP1:91,1] = PR[GP1:90,1] + 29.407;
   1:  PR[GP1:91,2] = PR[GP1:90,2] + 39.067;
   1:L PR[91] 10mm/sec CNT100;
   1:  PR[GP1:91,1] = PR[GP1:90,1] + 17.849;
   1:  PR[GP1:91,2] = PR[GP1:90,2] + 46.225;
   1:L PR[91] 10mm/sec CNT100;
   1:  PR[GP1:91,1] = PR[GP1:90,1] + 13.099;
   1:  PR[GP1:91,2] = PR[GP1:90,2] + 47.170;
   1:L PR[91] 10mm/sec CNT100;
   1:  PR[GP1:91,1] = PR[GP1:90,1] + -0.266;
   1:  PR[GP1:91,2] = PR[GP1:90,2] + 49.669;
   1:L PR[91] 10mm/sec CNT100;
   1:  PR[GP1:91,1] = PR[GP1:90,1] + -13.627;
   1:  PR[GP1:91,2] = PR[GP1:90,2] + 47.170;
   1:L PR[91] 10mm/sec CNT100;
   1:  PR[GP1:91,1] = PR[GP1:90,1] + -18.378;
   1:  PR[GP1:91,2] = PR[GP1:90,2] + 46.224;
   1:L PR[91] 10mm/sec CNT100;
   1:  PR[GP1:91,1] = PR[GP1:90,1] + -29.930;
   1:  PR[GP1:91,2] = PR[GP1:90,2] + 39.069;
   1:L PR[91] 10mm/sec CNT100;
   1:  PR[GP1:91,1] = PR[GP1:90,1] + -33.971;
   1:  PR[GP1:91,2] = PR[GP1:90,2] + 36.370;
   1:L PR[91] 10mm/sec CNT100;
   1:  PR[GP1:91,1] = PR[GP1:90,1] + -40.477;
   1:  PR[GP1:91,2] = PR[GP1:90,2] + 28.533;
   1:L PR[91] 10mm/sec CNT100;
   1:  PR[GP1:91,1] = PR[GP1:90,1] + -43.183;
   1:  PR[GP1:91,2] = PR[GP1:90,2] + 24.482;
   1:L PR[91] 10mm/sec CNT100;
   1:  PR[GP1:91,1] = PR[GP1:90,1] + -47.290;
   1:  PR[GP1:91,2] = PR[GP1:90,2] + 15.180;
   1:L PR[91] 10mm/sec CNT100;
   1:  PR[GP1:91,1] = PR[GP1:90,1] + -48.704;
   1:  PR[GP1:91,2] = PR[GP1:90,2] + 5.039;
   1:L PR[91] 10mm/sec CNT100;
   1:  PR[GP1:91,1] = PR[GP1:90,1] + -49.655;
   1:  PR[GP1:91,2] = PR[GP1:90,2] + 0.261;
   1:L PR[91] 10mm/sec CNT100;
   1:  PR[GP1:91,1] = PR[GP1:90,1] + -48.248;
   1:  PR[GP1:91,2] = PR[GP1:90,2] + -9.827;
   1:L PR[91] 10mm/sec CNT100;
   1:  PR[GP1:91,1] = PR[GP1:90,1] + -47.297;
   1:  PR[GP1:91,2] = PR[GP1:90,2] + -14.606;
   1:L PR[91] 10mm/sec CNT100;
   1:  PR[GP1:91,1] = PR[GP1:90,1] + -43.183;
   1:  PR[GP1:91,2] = PR[GP1:90,2] + -23.924;
   1:L PR[91] 10mm/sec CNT100;
   1:  PR[GP1:91,1] = PR[GP1:90,1] + -40.477;
   1:  PR[GP1:91,2] = PR[GP1:90,2] + -27.975;
   1:L PR[91] 10mm/sec CNT100;
   1:  PR[GP1:91,1] = PR[GP1:90,1] + -33.971;
   1:  PR[GP1:91,2] = PR[GP1:90,2] + -35.812;
   1:L PR[91] 10mm/sec CNT100;
   1:  PR[GP1:91,1] = PR[GP1:90,1] + -29.930;
   1:  PR[GP1:91,2] = PR[GP1:90,2] + -38.511;
   1:L PR[91] 10mm/sec CNT100;
   1:  PR[GP1:91,1] = PR[GP1:90,1] + -18.381;
   1:  PR[GP1:91,2] = PR[GP1:90,2] + -45.665;
   1:L PR[91] 10mm/sec CNT100;
   1:  PR[GP1:91,1] = PR[GP1:90,1] + -5.013;
   1:  PR[GP1:91,2] = PR[GP1:90,2] + -48.165;
   1:L PR[91] 10mm/sec CNT100;
   1:  PR[GP1:91,1] = PR[GP1:90,1] + -0.263;
   1:  PR[GP1:91,2] = PR[GP1:90,2] + -49.110;
   1:L PR[91] 10mm/sec CNT100;
   1:  PR[GP1:91,1] = PR[GP1:90,1] + 11.997;
   1:  PR[GP1:91,2] = PR[GP1:90,2] + -46.818;
   1:  PR[GP1:91,3] = PR[GP1:90,3] + 131.455;
   1:L PR[91] 10mm/sec CNT100;
   1:  PR[GP1:91,1] = PR[GP1:90,1] + 17.914;
   1:  PR[GP1:91,2] = PR[GP1:90,2] + -45.641;
   1:L PR[91] 10mm/sec CNT100;
   1:  PR[GP1:91,1] = PR[GP1:90,1] + 28.519;
   1:  PR[GP1:91,2] = PR[GP1:90,2] + -39.074;
   1:L PR[91] 10mm/sec CNT100;
   1:  PR[GP1:91,1] = PR[GP1:90,1] + 33.547;
   1:  PR[GP1:91,2] = PR[GP1:90,2] + -35.714;
   1:L PR[91] 10mm/sec CNT100;
   1:  PR[GP1:91,1] = PR[GP1:90,1] + 39.514;
   1:  PR[GP1:91,2] = PR[GP1:90,2] + -28.526;
   1:L PR[91] 10mm/sec CNT100;
   1:  PR[GP1:91,1] = PR[GP1:90,1] + 42.882;
   1:  PR[GP1:91,2] = PR[GP1:90,2] + -23.485;
   1:L PR[91] 10mm/sec CNT100;
   1:  PR[GP1:91,1] = PR[GP1:90,1] + 46.648;
   1:  PR[GP1:91,2] = PR[GP1:90,2] + -14.954;
   1:L PR[91] 10mm/sec CNT100;
   1:  PR[GP1:91,1] = PR[GP1:90,1] + 47.946;
   1:  PR[GP1:91,2] = PR[GP1:90,2] + -5.648;
   1:L PR[91] 10mm/sec CNT100;
   1:  PR[GP1:91,1] = PR[GP1:90,1] + 49.129;
   1:  PR[GP1:91,2] = PR[GP1:90,2] + 0.297;
   1:L PR[91] 10mm/sec CNT100;
   1:  PR[GP1:91,1] = PR[GP1:90,1] + 47.838;
   1:  PR[GP1:91,2] = PR[GP1:90,2] + 9.551;
   1:L PR[91] 10mm/sec CNT100;
   1:  PR[GP1:91,1] = PR[GP1:90,1] + 46.655;
   1:  PR[GP1:91,2] = PR[GP1:90,2] + 15.496;
   1:L PR[91] 10mm/sec CNT100;
   1:  PR[GP1:91,1] = PR[GP1:90,1] + 42.882;
   1:  PR[GP1:91,2] = PR[GP1:90,2] + 24.044;
   1:L PR[91] 10mm/sec CNT100;
   1:  PR[GP1:91,1] = PR[GP1:90,1] + 39.514;
   1:  PR[GP1:91,2] = PR[GP1:90,2] + 29.084;
   1:L PR[91] 10mm/sec CNT100;
   1:  PR[GP1:91,1] = PR[GP1:90,1] + 33.547;
   1:  PR[GP1:91,2] = PR[GP1:90,2] + 36.272;
   1:L PR[91] 10mm/sec CNT100;
   1:  PR[GP1:91,1] = PR[GP1:90,1] + 28.519;
   1:  PR[GP1:91,2] = PR[GP1:90,2] + 39.632;
   1:L PR[91] 10mm/sec CNT100;
   1:  PR[GP1:91,1] = PR[GP1:90,1] + 17.914;
   1:  PR[GP1:91,2] = PR[GP1:90,2] + 46.199;
   1:L PR[91] 10mm/sec CNT100;
   1:  PR[GP1:91,1] = PR[GP1:90,1] + 11.997;
   1:  PR[GP1:91,2] = PR[GP1:90,2] + 47.376;
   1:L PR[91] 10mm/sec CNT100;
   1:  PR[GP1:91,1] = PR[GP1:90,1] + -0.266;
   1:  PR[GP1:91,2] = PR[GP1:90,2] + 49.669;
   1:L PR[91] 10mm/sec CNT100;
   1:  PR[GP1:91,1] = PR[GP1:90,1] + -12.525;
   1:  PR[GP1:91,2] = PR[GP1:90,2] + 47.376;
   1:L PR[91] 10mm/sec CNT100;
   1:  PR[GP1:91,1] = PR[GP1:90,1] + -18.443;
   1:  PR[GP1:91,2] = PR[GP1:90,2] + 46.198;
   1:L PR[91] 10mm/sec CNT100;
   1:  PR[GP1:91,1] = PR[GP1:90,1] + -29.042;
   1:  PR[GP1:91,2] = PR[GP1:90,2] + 39.634;
   1:L PR[91] 10mm/sec CNT100;
   1:  PR[GP1:91,1] = PR[GP1:90,1] + -34.072;
   1:  PR[GP1:91,2] = PR[GP1:90,2] + 36.273;
   1:L PR[91] 10mm/sec CNT100;
   1:  PR[GP1:91,1] = PR[GP1:90,1] + -40.040;
   1:  PR[GP1:91,2] = PR[GP1:90,2] + 29.084;
   1:L PR[91] 10mm/sec CNT100;
   1:  PR[GP1:91,1] = PR[GP1:90,1] + -43.408;
   1:  PR[GP1:91,2] = PR[GP1:90,2] + 24.044;
   1:L PR[91] 10mm/sec CNT100;
   1:  PR[GP1:91,1] = PR[GP1:90,1] + -47.174;
   1:  PR[GP1:91,2] = PR[GP1:90,2] + 15.512;
   1:L PR[91] 10mm/sec CNT100;
   1:  PR[GP1:91,1] = PR[GP1:90,1] + -48.472;
   1:  PR[GP1:91,2] = PR[GP1:90,2] + 6.206;
   1:L PR[91] 10mm/sec CNT100;
   1:  PR[GP1:91,1] = PR[GP1:90,1] + -49.655;
   1:  PR[GP1:91,2] = PR[GP1:90,2] + 0.261;
   1:L PR[91] 10mm/sec CNT100;
   1:  PR[GP1:91,1] = PR[GP1:90,1] + -48.364;
   1:  PR[GP1:91,2] = PR[GP1:90,2] + -8.993;
   1:L PR[91] 10mm/sec CNT100;
   1:  PR[GP1:91,1] = PR[GP1:90,1] + -47.181;
   1:  PR[GP1:91,2] = PR[GP1:90,2] + -14.938;
   1:L PR[91] 10mm/sec CNT100;
   1:  PR[GP1:91,1] = PR[GP1:90,1] + -43.408;
   1:  PR[GP1:91,2] = PR[GP1:90,2] + -23.486;
   1:L PR[91] 10mm/sec CNT100;
   1:  PR[GP1:91,1] = PR[GP1:90,1] + -40.040;
   1:  PR[GP1:91,2] = PR[GP1:90,2] + -28.526;
   1:L PR[91] 10mm/sec CNT100;
   1:  PR[GP1:91,1] = PR[GP1:90,1] + -34.072;
   1:  PR[GP1:91,2] = PR[GP1:90,2] + -35.715;
   1:L PR[91] 10mm/sec CNT100;
   1:  PR[GP1:91,1] = PR[GP1:90,1] + -29.042;
   1:  PR[GP1:91,2] = PR[GP1:90,2] + -39.075;
   1:L PR[91] 10mm/sec CNT100;
   1:  PR[GP1:91,1] = PR[GP1:90,1] + -18.446;
   1:  PR[GP1:91,2] = PR[GP1:90,2] + -45.638;
   1:L PR[91] 10mm/sec CNT100;
   1:  PR[GP1:91,1] = PR[GP1:90,1] + -6.180;
   1:  PR[GP1:91,2] = PR[GP1:90,2] + -47.933;
   1:L PR[91] 10mm/sec CNT100;
   1:  PR[GP1:91,1] = PR[GP1:90,1] + -0.263;
   1:  PR[GP1:91,2] = PR[GP1:90,2] + -49.110;
   1:L PR[91] 10mm/sec CNT100;
   1:  PR[GP1:91,1] = PR[GP1:90,1] + 10.895;
   1:  PR[GP1:91,2] = PR[GP1:90,2] + -47.024;
   1:  PR[GP1:91,3] = PR[GP1:90,3] + 132.065;
   1:L PR[91] 10mm/sec CNT100;
   1:  PR[GP1:91,1] = PR[GP1:90,1] + 17.980;
   1:  PR[GP1:91,2] = PR[GP1:90,2] + -45.615;
   1:L PR[91] 10mm/sec CNT100;
   1:  PR[GP1:91,1] = PR[GP1:90,1] + 27.631;
   1:  PR[GP1:91,2] = PR[GP1:90,2] + -39.638;
   1:L PR[91] 10mm/sec CNT100;
   1:  PR[GP1:91,1] = PR[GP1:90,1] + 33.648;
   1:  PR[GP1:91,2] = PR[GP1:90,2] + -35.617;
   1:L PR[91] 10mm/sec CNT100;
   1:  PR[GP1:91,1] = PR[GP1:90,1] + 39.077;
   1:  PR[GP1:91,2] = PR[GP1:90,2] + -29.077;
   1:L PR[91] 10mm/sec CNT100;
   1:  PR[GP1:91,1] = PR[GP1:90,1] + 43.106;
   1:  PR[GP1:91,2] = PR[GP1:90,2] + -23.047;
   1:L PR[91] 10mm/sec CNT100;
   1:  PR[GP1:91,1] = PR[GP1:90,1] + 46.532;
   1:  PR[GP1:91,2] = PR[GP1:90,2] + -15.287;
   1:L PR[91] 10mm/sec CNT100;
   1:  PR[GP1:91,1] = PR[GP1:90,1] + 47.714;
   1:  PR[GP1:91,2] = PR[GP1:90,2] + -6.815;
   1:L PR[91] 10mm/sec CNT100;
   1:  PR[GP1:91,1] = PR[GP1:90,1] + 49.129;
   1:  PR[GP1:91,2] = PR[GP1:90,2] + 0.297;
   1:L PR[91] 10mm/sec CNT100;
   1:  PR[GP1:91,1] = PR[GP1:90,1] + 47.954;
   1:  PR[GP1:91,2] = PR[GP1:90,2] + 8.716;
   1:L PR[91] 10mm/sec CNT100;
   1:  PR[GP1:91,1] = PR[GP1:90,1] + 46.539;
   1:  PR[GP1:91,2] = PR[GP1:90,2] + 15.828;
   1:L PR[91] 10mm/sec CNT100;
   1:  PR[GP1:91,1] = PR[GP1:90,1] + 43.106;
   1:  PR[GP1:91,2] = PR[GP1:90,2] + 23.605;
   1:L PR[91] 10mm/sec CNT100;
   1:  PR[GP1:91,1] = PR[GP1:90,1] + 39.077;
   1:  PR[GP1:91,2] = PR[GP1:90,2] + 29.635;
   1:L PR[91] 10mm/sec CNT100;
   1:  PR[GP1:91,1] = PR[GP1:90,1] + 33.648;
   1:  PR[GP1:91,2] = PR[GP1:90,2] + 36.175;
   1:L PR[91] 10mm/sec CNT100;
   1:  PR[GP1:91,1] = PR[GP1:90,1] + 27.631;
   1:  PR[GP1:91,2] = PR[GP1:90,2] + 40.196;
   1:L PR[91] 10mm/sec CNT100;
   1:  PR[GP1:91,1] = PR[GP1:90,1] + 17.980;
   1:  PR[GP1:91,2] = PR[GP1:90,2] + 46.173;
   1:L PR[91] 10mm/sec CNT100;
   1:  PR[GP1:91,1] = PR[GP1:90,1] + 10.895;
   1:  PR[GP1:91,2] = PR[GP1:90,2] + 47.582;
   1:L PR[91] 10mm/sec CNT100;
   1:  PR[GP1:91,1] = PR[GP1:90,1] + -0.266;
   1:  PR[GP1:91,2] = PR[GP1:90,2] + 49.669;
   1:L PR[91] 10mm/sec CNT100;
   1:  PR[GP1:91,1] = PR[GP1:90,1] + -11.423;
   1:  PR[GP1:91,2] = PR[GP1:90,2] + 47.582;
   1:L PR[91] 10mm/sec CNT100;
   1:  PR[GP1:91,1] = PR[GP1:90,1] + -18.508;
   1:  PR[GP1:91,2] = PR[GP1:90,2] + 46.172;
   1:L PR[91] 10mm/sec CNT100;
   1:  PR[GP1:91,1] = PR[GP1:90,1] + -28.155;
   1:  PR[GP1:91,2] = PR[GP1:90,2] + 40.198;
   1:L PR[91] 10mm/sec CNT100;
   1:  PR[GP1:91,1] = PR[GP1:90,1] + -34.174;
   1:  PR[GP1:91,2] = PR[GP1:90,2] + 36.176;
   1:L PR[91] 10mm/sec CNT100;
   1:  PR[GP1:91,1] = PR[GP1:90,1] + -39.603;
   1:  PR[GP1:91,2] = PR[GP1:90,2] + 29.636;
   1:L PR[91] 10mm/sec CNT100;
   1:  PR[GP1:91,1] = PR[GP1:90,1] + -43.632;
   1:  PR[GP1:91,2] = PR[GP1:90,2] + 23.606;
   1:L PR[91] 10mm/sec CNT100;
   1:  PR[GP1:91,1] = PR[GP1:90,1] + -47.058;
   1:  PR[GP1:91,2] = PR[GP1:90,2] + 15.845;
   1:L PR[91] 10mm/sec CNT100;
   1:  PR[GP1:91,1] = PR[GP1:90,1] + -48.240;
   1:  PR[GP1:91,2] = PR[GP1:90,2] + 7.373;
   1:L PR[91] 10mm/sec CNT100;
   1:  PR[GP1:91,1] = PR[GP1:90,1] + -49.655;
   1:  PR[GP1:91,2] = PR[GP1:90,2] + 0.261;
   1:L PR[91] 10mm/sec CNT100;
   1:  PR[GP1:91,1] = PR[GP1:90,1] + -48.481;
   1:  PR[GP1:91,2] = PR[GP1:90,2] + -8.158;
   1:L PR[91] 10mm/sec CNT100;
   1:  PR[GP1:91,1] = PR[GP1:90,1] + -47.066;
   1:  PR[GP1:91,2] = PR[GP1:90,2] + -15.271;
   1:L PR[91] 10mm/sec CNT100;
   1:  PR[GP1:91,1] = PR[GP1:90,1] + -43.632;
   1:  PR[GP1:91,2] = PR[GP1:90,2] + -23.048;
   1:L PR[91] 10mm/sec CNT100;
   1:  PR[GP1:91,1] = PR[GP1:90,1] + -39.603;
   1:  PR[GP1:91,2] = PR[GP1:90,2] + -29.078;
   1:L PR[91] 10mm/sec CNT100;
   1:  PR[GP1:91,1] = PR[GP1:90,1] + -34.174;
   1:  PR[GP1:91,2] = PR[GP1:90,2] + -35.618;
   1:L PR[91] 10mm/sec CNT100;
   1:  PR[GP1:91,1] = PR[GP1:90,1] + -28.155;
   1:  PR[GP1:91,2] = PR[GP1:90,2] + -39.639;
   1:L PR[91] 10mm/sec CNT100;
   1:  PR[GP1:91,1] = PR[GP1:90,1] + -18.511;
   1:  PR[GP1:91,2] = PR[GP1:90,2] + -45.612;
   1:L PR[91] 10mm/sec CNT100;
   1:  PR[GP1:91,1] = PR[GP1:90,1] + -7.346;
   1:  PR[GP1:91,2] = PR[GP1:90,2] + -47.700;
   1:L PR[91] 10mm/sec CNT100;
   1:  PR[GP1:91,1] = PR[GP1:90,1] + -0.262;
   1:  PR[GP1:91,2] = PR[GP1:90,2] + -49.110;
   1:L PR[91] 10mm/sec CNT100;
   1:  PR[GP1:91,1] = PR[GP1:90,1] + 9.793;
   1:  PR[GP1:91,2] = PR[GP1:90,2] + -47.230;
   1:  PR[GP1:91,3] = PR[GP1:90,3] + 132.675;
   1:L PR[91] 10mm/sec CNT100;
   1:  PR[GP1:91,1] = PR[GP1:90,1] + 18.045;
   1:  PR[GP1:91,2] = PR[GP1:90,2] + -45.589;
   1:L PR[91] 10mm/sec CNT100;
   1:  PR[GP1:91,1] = PR[GP1:90,1] + 26.743;
   1:  PR[GP1:91,2] = PR[GP1:90,2] + -40.202;
   1:L PR[91] 10mm/sec CNT100;
   1:  PR[GP1:91,1] = PR[GP1:90,1] + 33.750;
   1:  PR[GP1:91,2] = PR[GP1:90,2] + -35.520;
   1:L PR[91] 10mm/sec CNT100;
   1:  PR[GP1:91,1] = PR[GP1:90,1] + 38.641;
   1:  PR[GP1:91,2] = PR[GP1:90,2] + -29.628;
   1:L PR[91] 10mm/sec CNT100;
   1:  PR[GP1:91,1] = PR[GP1:90,1] + 43.331;
   1:  PR[GP1:91,2] = PR[GP1:90,2] + -22.609;
   1:L PR[91] 10mm/sec CNT100;
   1:  PR[GP1:91,1] = PR[GP1:90,1] + 46.416;
   1:  PR[GP1:91,2] = PR[GP1:90,2] + -15.619;
   1:L PR[91] 10mm/sec CNT100;
   1:  PR[GP1:91,1] = PR[GP1:90,1] + 47.481;
   1:  PR[GP1:91,2] = PR[GP1:90,2] + -7.982;
   1:L PR[91] 10mm/sec CNT100;
   1:  PR[GP1:91,1] = PR[GP1:90,1] + 49.129;
   1:  PR[GP1:91,2] = PR[GP1:90,2] + 0.297;
   1:L PR[91] 10mm/sec CNT100;
   1:  PR[GP1:91,1] = PR[GP1:90,1] + 48.071;
   1:  PR[GP1:91,2] = PR[GP1:90,2] + 7.882;
   1:L PR[91] 10mm/sec CNT100;
   1:  PR[GP1:91,1] = PR[GP1:90,1] + 46.423;
   1:  PR[GP1:91,2] = PR[GP1:90,2] + 16.161;
   1:L PR[91] 10mm/sec CNT100;
   1:  PR[GP1:91,1] = PR[GP1:90,1] + 43.331;
   1:  PR[GP1:91,2] = PR[GP1:90,2] + 23.167;
   1:L PR[91] 10mm/sec CNT100;
   1:  PR[GP1:91,1] = PR[GP1:90,1] + 38.641;
   1:  PR[GP1:91,2] = PR[GP1:90,2] + 30.186;
   1:L PR[91] 10mm/sec CNT100;
   1:  PR[GP1:91,1] = PR[GP1:90,1] + 33.750;
   1:  PR[GP1:91,2] = PR[GP1:90,2] + 36.079;
   1:L PR[91] 10mm/sec CNT100;
   1:  PR[GP1:91,1] = PR[GP1:90,1] + 26.743;
   1:  PR[GP1:91,2] = PR[GP1:90,2] + 40.760;
   1:L PR[91] 10mm/sec CNT100;
   1:  PR[GP1:91,1] = PR[GP1:90,1] + 18.045;
   1:  PR[GP1:91,2] = PR[GP1:90,2] + 46.147;
   1:L PR[91] 10mm/sec CNT100;
   1:  PR[GP1:91,1] = PR[GP1:90,1] + 9.793;
   1:  PR[GP1:91,2] = PR[GP1:90,2] + 47.788;
   1:L PR[91] 10mm/sec CNT100;
   1:  PR[GP1:91,1] = PR[GP1:90,1] + -0.266;
   1:  PR[GP1:91,2] = PR[GP1:90,2] + 49.669;
   1:L PR[91] 10mm/sec CNT100;
   1:  PR[GP1:91,1] = PR[GP1:90,1] + -10.321;
   1:  PR[GP1:91,2] = PR[GP1:90,2] + 47.788;
   1:L PR[91] 10mm/sec CNT100;
   1:  PR[GP1:91,1] = PR[GP1:90,1] + -18.573;
   1:  PR[GP1:91,2] = PR[GP1:90,2] + 46.146;
   1:L PR[91] 10mm/sec CNT100;
   1:  PR[GP1:91,1] = PR[GP1:90,1] + -27.267;
   1:  PR[GP1:91,2] = PR[GP1:90,2] + 40.762;
   1:L PR[91] 10mm/sec CNT100;
   1:  PR[GP1:91,1] = PR[GP1:90,1] + -34.275;
   1:  PR[GP1:91,2] = PR[GP1:90,2] + 36.079;
   1:L PR[91] 10mm/sec CNT100;
   1:  PR[GP1:91,1] = PR[GP1:90,1] + -39.167;
   1:  PR[GP1:91,2] = PR[GP1:90,2] + 30.187;
   1:L PR[91] 10mm/sec CNT100;
   1:  PR[GP1:91,1] = PR[GP1:90,1] + -43.857;
   1:  PR[GP1:91,2] = PR[GP1:90,2] + 23.168;
   1:L PR[91] 10mm/sec CNT100;
   1:  PR[GP1:91,1] = PR[GP1:90,1] + -46.943;
   1:  PR[GP1:91,2] = PR[GP1:90,2] + 16.177;
   1:L PR[91] 10mm/sec CNT100;
   1:  PR[GP1:91,1] = PR[GP1:90,1] + -48.008;
   1:  PR[GP1:91,2] = PR[GP1:90,2] + 8.540;
   1:L PR[91] 10mm/sec CNT100;
   1:  PR[GP1:91,1] = PR[GP1:90,1] + -49.655;
   1:  PR[GP1:91,2] = PR[GP1:90,2] + 0.261;
   1:L PR[91] 10mm/sec CNT100;
   1:  PR[GP1:91,1] = PR[GP1:90,1] + -48.597;
   1:  PR[GP1:91,2] = PR[GP1:90,2] + -7.324;
   1:L PR[91] 10mm/sec CNT100;
   1:  PR[GP1:91,1] = PR[GP1:90,1] + -46.950;
   1:  PR[GP1:91,2] = PR[GP1:90,2] + -15.603;
   1:L PR[91] 10mm/sec CNT100;
   1:  PR[GP1:91,1] = PR[GP1:90,1] + -43.857;
   1:  PR[GP1:91,2] = PR[GP1:90,2] + -22.610;
   1:L PR[91] 10mm/sec CNT100;
   1:  PR[GP1:91,1] = PR[GP1:90,1] + -39.167;
   1:  PR[GP1:91,2] = PR[GP1:90,2] + -29.629;
   1:L PR[91] 10mm/sec CNT100;
   1:  PR[GP1:91,1] = PR[GP1:90,1] + -34.275;
   1:  PR[GP1:91,2] = PR[GP1:90,2] + -35.521;
   1:L PR[91] 10mm/sec CNT100;
   1:  PR[GP1:91,1] = PR[GP1:90,1] + -27.267;
   1:  PR[GP1:91,2] = PR[GP1:90,2] + -40.204;
   1:L PR[91] 10mm/sec CNT100;
   1:  PR[GP1:91,1] = PR[GP1:90,1] + -18.576;
   1:  PR[GP1:91,2] = PR[GP1:90,2] + -45.586;
   1:L PR[91] 10mm/sec CNT100;
   1:  PR[GP1:91,1] = PR[GP1:90,1] + -8.513;
   1:  PR[GP1:91,2] = PR[GP1:90,2] + -47.468;
   1:L PR[91] 10mm/sec CNT100;
   1:  PR[GP1:91,1] = PR[GP1:90,1] + -0.262;
   1:  PR[GP1:91,2] = PR[GP1:90,2] + -49.110;
   1:L PR[91] 10mm/sec CNT100;
   1:  PR[GP1:91,1] = PR[GP1:90,1] + 8.691;
   1:  PR[GP1:91,2] = PR[GP1:90,2] + -47.436;
   1:  PR[GP1:91,3] = PR[GP1:90,3] + 133.285;
   1:L PR[91] 10mm/sec CNT100;
   1:  PR[GP1:91,1] = PR[GP1:90,1] + 18.110;
   1:  PR[GP1:91,2] = PR[GP1:90,2] + -45.563;
   1:L PR[91] 10mm/sec CNT100;
   1:  PR[GP1:91,1] = PR[GP1:90,1] + 25.855;
   1:  PR[GP1:91,2] = PR[GP1:90,2] + -40.766;
   1:L PR[91] 10mm/sec CNT100;
   1:  PR[GP1:91,1] = PR[GP1:90,1] + 33.851;
   1:  PR[GP1:91,2] = PR[GP1:90,2] + -35.424;
   1:L PR[91] 10mm/sec CNT100;
   1:  PR[GP1:91,1] = PR[GP1:90,1] + 38.204;
   1:  PR[GP1:91,2] = PR[GP1:90,2] + -30.180;
   1:L PR[91] 10mm/sec CNT100;
   1:  PR[GP1:91,1] = PR[GP1:90,1] + 43.555;
   1:  PR[GP1:91,2] = PR[GP1:90,2] + -22.171;
   1:L PR[91] 10mm/sec CNT100;
   1:  PR[GP1:91,1] = PR[GP1:90,1] + 46.301;
   1:  PR[GP1:91,2] = PR[GP1:90,2] + -15.952;
   1:L PR[91] 10mm/sec CNT100;
   1:  PR[GP1:91,1] = PR[GP1:90,1] + 47.249;
   1:  PR[GP1:91,2] = PR[GP1:90,2] + -9.149;
   1:L PR[91] 10mm/sec CNT100;
   1:  PR[GP1:91,1] = PR[GP1:90,1] + 49.129;
   1:  PR[GP1:91,2] = PR[GP1:90,2] + 0.297;
   1:L PR[91] 10mm/sec CNT100;
   1:  PR[GP1:91,1] = PR[GP1:90,1] + 48.187;
   1:  PR[GP1:91,2] = PR[GP1:90,2] + 7.047;
   1:L PR[91] 10mm/sec CNT100;
   1:  PR[GP1:91,1] = PR[GP1:90,1] + 46.308;
   1:  PR[GP1:91,2] = PR[GP1:90,2] + 16.494;
   1:L PR[91] 10mm/sec CNT100;
   1:  PR[GP1:91,1] = PR[GP1:90,1] + 43.555;
   1:  PR[GP1:91,2] = PR[GP1:90,2] + 22.729;
   1:L PR[91] 10mm/sec CNT100;
   1:  PR[GP1:91,1] = PR[GP1:90,1] + 38.204;
   1:  PR[GP1:91,2] = PR[GP1:90,2] + 30.738;
   1:L PR[91] 10mm/sec CNT100;
   1:  PR[GP1:91,1] = PR[GP1:90,1] + 33.851;
   1:  PR[GP1:91,2] = PR[GP1:90,2] + 35.982;
   1:L PR[91] 10mm/sec CNT100;
   1:  PR[GP1:91,1] = PR[GP1:90,1] + 25.855;
   1:  PR[GP1:91,2] = PR[GP1:90,2] + 41.324;
   1:L PR[91] 10mm/sec CNT100;
   1:  PR[GP1:91,1] = PR[GP1:90,1] + 18.110;
   1:  PR[GP1:91,2] = PR[GP1:90,2] + 46.121;
   1:L PR[91] 10mm/sec CNT100;
   1:  PR[GP1:91,1] = PR[GP1:90,1] + 8.691;
   1:  PR[GP1:91,2] = PR[GP1:90,2] + 47.994;
   1:L PR[91] 10mm/sec CNT100;
   1:  PR[GP1:91,1] = PR[GP1:90,1] + -0.265;
   1:  PR[GP1:91,2] = PR[GP1:90,2] + 49.669;
   1:L PR[91] 10mm/sec CNT100;
   1:  PR[GP1:91,1] = PR[GP1:90,1] + -9.219;
   1:  PR[GP1:91,2] = PR[GP1:90,2] + 47.994;
   1:L PR[91] 10mm/sec CNT100;
   1:  PR[GP1:91,1] = PR[GP1:90,1] + -18.638;
   1:  PR[GP1:91,2] = PR[GP1:90,2] + 46.120;
   1:L PR[91] 10mm/sec CNT100;
   1:  PR[GP1:91,1] = PR[GP1:90,1] + -26.379;
   1:  PR[GP1:91,2] = PR[GP1:90,2] + 41.326;
   1:L PR[91] 10mm/sec CNT100;
   1:  PR[GP1:91,1] = PR[GP1:90,1] + -34.377;
   1:  PR[GP1:91,2] = PR[GP1:90,2] + 35.982;
   1:L PR[91] 10mm/sec CNT100;
   1:  PR[GP1:91,1] = PR[GP1:90,1] + -38.730;
   1:  PR[GP1:91,2] = PR[GP1:90,2] + 30.738;
   1:L PR[91] 10mm/sec CNT100;
   1:  PR[GP1:91,1] = PR[GP1:90,1] + -44.081;
   1:  PR[GP1:91,2] = PR[GP1:90,2] + 22.729;
   1:L PR[91] 10mm/sec CNT100;
   1:  PR[GP1:91,1] = PR[GP1:90,1] + -46.827;
   1:  PR[GP1:91,2] = PR[GP1:90,2] + 16.510;
   1:L PR[91] 10mm/sec CNT100;
   1:  PR[GP1:91,1] = PR[GP1:90,1] + -47.776;
   1:  PR[GP1:91,2] = PR[GP1:90,2] + 9.707;
   1:L PR[91] 10mm/sec CNT100;
   1:  PR[GP1:91,1] = PR[GP1:90,1] + -49.655;
   1:  PR[GP1:91,2] = PR[GP1:90,2] + 0.261;
   1:L PR[91] 10mm/sec CNT100;
   1:  PR[GP1:91,1] = PR[GP1:90,1] + -48.713;
   1:  PR[GP1:91,2] = PR[GP1:90,2] + -6.489;
   1:L PR[91] 10mm/sec CNT100;
   1:  PR[GP1:91,1] = PR[GP1:90,1] + -46.834;
   1:  PR[GP1:91,2] = PR[GP1:90,2] + -15.936;
   1:L PR[91] 10mm/sec CNT100;
   1:  PR[GP1:91,1] = PR[GP1:90,1] + -44.081;
   1:  PR[GP1:91,2] = PR[GP1:90,2] + -22.171;
   1:L PR[91] 10mm/sec CNT100;
   1:  PR[GP1:91,1] = PR[GP1:90,1] + -38.730;
   1:  PR[GP1:91,2] = PR[GP1:90,2] + -30.180;
   1:L PR[91] 10mm/sec CNT100;
   1:  PR[GP1:91,1] = PR[GP1:90,1] + -34.377;
   1:  PR[GP1:91,2] = PR[GP1:90,2] + -35.424;
   1:L PR[91] 10mm/sec CNT100;
   1:  PR[GP1:91,1] = PR[GP1:90,1] + -26.379;
   1:  PR[GP1:91,2] = PR[GP1:90,2] + -40.768;
   1:L PR[91] 10mm/sec CNT100;
   1:  PR[GP1:91,1] = PR[GP1:90,1] + -18.641;
   1:  PR[GP1:91,2] = PR[GP1:90,2] + -45.560;
   1:L PR[91] 10mm/sec CNT100;
   1:  PR[GP1:91,1] = PR[GP1:90,1] + -9.680;
   1:  PR[GP1:91,2] = PR[GP1:90,2] + -47.236;
   1:L PR[91] 10mm/sec CNT100;
   1:  PR[GP1:91,1] = PR[GP1:90,1] + -0.262;
   1:  PR[GP1:91,2] = PR[GP1:90,2] + -49.110;
   1:L PR[91] 10mm/sec CNT100;
   1:  PR[GP1:91,1] = PR[GP1:90,1] + 7.589;
   1:  PR[GP1:91,2] = PR[GP1:90,2] + -47.642;
   1:  PR[GP1:91,3] = PR[GP1:90,3] + 133.895;
   1:L PR[91] 10mm/sec CNT100;
   1:  PR[GP1:91,1] = PR[GP1:90,1] + 18.175;
   1:  PR[GP1:91,2] = PR[GP1:90,2] + -45.536;
   1:L PR[91] 10mm/sec CNT100;
   1:  PR[GP1:91,1] = PR[GP1:90,1] + 24.966;
   1:  PR[GP1:91,2] = PR[GP1:90,2] + -41.330;
   1:L PR[91] 10mm/sec CNT100;
   1:  PR[GP1:91,1] = PR[GP1:90,1] + 33.952;
   1:  PR[GP1:91,2] = PR[GP1:90,2] + -35.327;
   1:L PR[91] 10mm/sec CNT100;
   1:  PR[GP1:91,1] = PR[GP1:90,1] + 37.767;
   1:  PR[GP1:91,2] = PR[GP1:90,2] + -30.731;
   1:L PR[91] 10mm/sec CNT100;
   1:  PR[GP1:91,1] = PR[GP1:90,1] + 43.780;
   1:  PR[GP1:91,2] = PR[GP1:90,2] + -21.733;
   1:L PR[91] 10mm/sec CNT100;
   1:  PR[GP1:91,1] = PR[GP1:90,1] + 46.185;
   1:  PR[GP1:91,2] = PR[GP1:90,2] + -16.284;
   1:L PR[91] 10mm/sec CNT100;
   1:  PR[GP1:91,1] = PR[GP1:90,1] + 47.017;
   1:  PR[GP1:91,2] = PR[GP1:90,2] + -10.317;
   1:L PR[91] 10mm/sec CNT100;
   1:  PR[GP1:91,1] = PR[GP1:90,1] + 49.129;
   1:  PR[GP1:91,2] = PR[GP1:90,2] + 0.297;
   1:L PR[91] 10mm/sec CNT100;
   1:  PR[GP1:91,1] = PR[GP1:90,1] + 48.303;
   1:  PR[GP1:91,2] = PR[GP1:90,2] + 6.212;
   1:L PR[91] 10mm/sec CNT100;
   1:  PR[GP1:91,1] = PR[GP1:90,1] + 46.192;
   1:  PR[GP1:91,2] = PR[GP1:90,2] + 16.826;
   1:L PR[91] 10mm/sec CNT100;
   1:  PR[GP1:91,1] = PR[GP1:90,1] + 43.780;
   1:  PR[GP1:91,2] = PR[GP1:90,2] + 22.291;
   1:L PR[91] 10mm/sec CNT100;
   1:  PR[GP1:91,1] = PR[GP1:90,1] + 37.767;
   1:  PR[GP1:91,2] = PR[GP1:90,2] + 31.289;
   1:L PR[91] 10mm/sec CNT100;
   1:  PR[GP1:91,1] = PR[GP1:90,1] + 33.952;
   1:  PR[GP1:91,2] = PR[GP1:90,2] + 35.885;
   1:L PR[91] 10mm/sec CNT100;
   1:  PR[GP1:91,1] = PR[GP1:90,1] + 24.966;
   1:  PR[GP1:91,2] = PR[GP1:90,2] + 41.889;
   1:L PR[91] 10mm/sec CNT100;
   1:  PR[GP1:91,1] = PR[GP1:90,1] + 18.175;
   1:  PR[GP1:91,2] = PR[GP1:90,2] + 46.094;
   1:L PR[91] 10mm/sec CNT100;
   1:  PR[GP1:91,1] = PR[GP1:90,1] + 7.590;
   1:  PR[GP1:91,2] = PR[GP1:90,2] + 48.200;
   1:L PR[91] 10mm/sec CNT100;
   1:  PR[GP1:91,1] = PR[GP1:90,1] + -0.265;
   1:  PR[GP1:91,2] = PR[GP1:90,2] + 49.669;
   1:L PR[91] 10mm/sec CNT100;
   1:  PR[GP1:91,1] = PR[GP1:90,1] + -8.117;
   1:  PR[GP1:91,2] = PR[GP1:90,2] + 48.200;
   1:L PR[91] 10mm/sec CNT100;
   1:  PR[GP1:91,1] = PR[GP1:90,1] + -18.703;
   1:  PR[GP1:91,2] = PR[GP1:90,2] + 46.094;
   1:L PR[91] 10mm/sec CNT100;
   1:  PR[GP1:91,1] = PR[GP1:90,1] + -25.491;
   1:  PR[GP1:91,2] = PR[GP1:90,2] + 41.890;
   1:L PR[91] 10mm/sec CNT100;
   1:  PR[GP1:91,1] = PR[GP1:90,1] + -34.479;
   1:  PR[GP1:91,2] = PR[GP1:90,2] + 35.885;
   1:L PR[91] 10mm/sec CNT100;
   1:  PR[GP1:91,1] = PR[GP1:90,1] + -38.294;
   1:  PR[GP1:91,2] = PR[GP1:90,2] + 31.290;
   1:L PR[91] 10mm/sec CNT100;
   1:  PR[GP1:91,1] = PR[GP1:90,1] + -44.306;
   1:  PR[GP1:91,2] = PR[GP1:90,2] + 22.291;
   1:L PR[91] 10mm/sec CNT100;
   1:  PR[GP1:91,1] = PR[GP1:90,1] + -46.711;
   1:  PR[GP1:91,2] = PR[GP1:90,2] + 16.843;
   1:L PR[91] 10mm/sec CNT100;
   1:  PR[GP1:91,1] = PR[GP1:90,1] + -47.543;
   1:  PR[GP1:91,2] = PR[GP1:90,2] + 10.875;
   1:L PR[91] 10mm/sec CNT100;
   1:  PR[GP1:91,1] = PR[GP1:90,1] + -49.655;
   1:  PR[GP1:91,2] = PR[GP1:90,2] + 0.261;
   1:L PR[91] 10mm/sec CNT100;
   1:  PR[GP1:91,1] = PR[GP1:90,1] + -48.830;
   1:  PR[GP1:91,2] = PR[GP1:90,2] + -5.655;
   1:L PR[91] 10mm/sec CNT100;
   1:  PR[GP1:91,1] = PR[GP1:90,1] + -46.718;
   1:  PR[GP1:91,2] = PR[GP1:90,2] + -16.268;
   1:L PR[91] 10mm/sec CNT100;
   1:  PR[GP1:91,1] = PR[GP1:90,1] + -44.306;
   1:  PR[GP1:91,2] = PR[GP1:90,2] + -21.733;
   1:L PR[91] 10mm/sec CNT100;
   1:  PR[GP1:91,1] = PR[GP1:90,1] + -38.294;
   1:  PR[GP1:91,2] = PR[GP1:90,2] + -30.731;
   1:L PR[91] 10mm/sec CNT100;
   1:  PR[GP1:91,1] = PR[GP1:90,1] + -34.479;
   1:  PR[GP1:91,2] = PR[GP1:90,2] + -35.327;
   1:L PR[91] 10mm/sec CNT100;
   1:  PR[GP1:91,1] = PR[GP1:90,1] + -25.491;
   1:  PR[GP1:91,2] = PR[GP1:90,2] + -41.332;
   1:L PR[91] 10mm/sec CNT100;
   1:  PR[GP1:91,1] = PR[GP1:90,1] + -18.706;
   1:  PR[GP1:91,2] = PR[GP1:90,2] + -45.534;
   1:L PR[91] 10mm/sec CNT100;
   1:  PR[GP1:91,1] = PR[GP1:90,1] + -10.847;
   1:  PR[GP1:91,2] = PR[GP1:90,2] + -47.004;
   1:L PR[91] 10mm/sec CNT100;
   1:  PR[GP1:91,1] = PR[GP1:90,1] + -0.261;
   1:  PR[GP1:91,2] = PR[GP1:90,2] + -49.110;
   1:L PR[91] 10mm/sec CNT100;
   1:  PR[GP1:91,1] = PR[GP1:90,1] + 6.487;
   1:  PR[GP1:91,2] = PR[GP1:90,2] + -47.848;
   1:  PR[GP1:91,3] = PR[GP1:90,3] + 134.505;
   1:L PR[91] 10mm/sec CNT100;
   1:  PR[GP1:91,1] = PR[GP1:90,1] + 18.241;
   1:  PR[GP1:91,2] = PR[GP1:90,2] + -45.510;
   1:L PR[91] 10mm/sec CNT100;
   1:  PR[GP1:91,1] = PR[GP1:90,1] + 24.078;
   1:  PR[GP1:91,2] = PR[GP1:90,2] + -41.895;
   1:L PR[91] 10mm/sec CNT100;
   1:  PR[GP1:91,1] = PR[GP1:90,1] + 34.054;
   1:  PR[GP1:91,2] = PR[GP1:90,2] + -35.230;
   1:L PR[91] 10mm/sec CNT100;
   1:  PR[GP1:91,1] = PR[GP1:90,1] + 37.331;
   1:  PR[GP1:91,2] = PR[GP1:90,2] + -31.282;
   1:L PR[91] 10mm/sec CNT100;
   1:  PR[GP1:91,1] = PR[GP1:90,1] + 44.004;
   1:  PR[GP1:91,2] = PR[GP1:90,2] + -21.295;
   1:L PR[91] 10mm/sec CNT100;
   1:  PR[GP1:91,1] = PR[GP1:90,1] + 46.069;
   1:  PR[GP1:91,2] = PR[GP1:90,2] + -16.617;
   1:L PR[91] 10mm/sec CNT100;
   1:  PR[GP1:91,1] = PR[GP1:90,1] + 46.785;
   1:  PR[GP1:91,2] = PR[GP1:90,2] + -11.484;
   1:L PR[91] 10mm/sec CNT100;
   1:  PR[GP1:91,1] = PR[GP1:90,1] + 49.129;
   1:  PR[GP1:91,2] = PR[GP1:90,2] + 0.297;
   1:L PR[91] 10mm/sec CNT100;
   1:  PR[GP1:91,1] = PR[GP1:90,1] + 48.420;
   1:  PR[GP1:91,2] = PR[GP1:90,2] + 5.378;
   1:L PR[91] 10mm/sec CNT100;
   1:  PR[GP1:91,1] = PR[GP1:90,1] + 46.076;
   1:  PR[GP1:91,2] = PR[GP1:90,2] + 17.159;
   1:L PR[91] 10mm/sec CNT100;
   1:  PR[GP1:91,1] = PR[GP1:90,1] + 44.004;
   1:  PR[GP1:91,2] = PR[GP1:90,2] + 21.853;
   1:L PR[91] 10mm/sec CNT100;
   1:  PR[GP1:91,1] = PR[GP1:90,1] + 37.331;
   1:  PR[GP1:91,2] = PR[GP1:90,2] + 31.840;
   1:L PR[91] 10mm/sec CNT100;
   1:  PR[GP1:91,1] = PR[GP1:90,1] + 34.054;
   1:  PR[GP1:91,2] = PR[GP1:90,2] + 35.788;
   1:L PR[91] 10mm/sec CNT100;
   1:  PR[GP1:91,1] = PR[GP1:90,1] + 24.078;
   1:  PR[GP1:91,2] = PR[GP1:90,2] + 42.453;
   1:L PR[91] 10mm/sec CNT100;
   1:  PR[GP1:91,1] = PR[GP1:90,1] + 18.241;
   1:  PR[GP1:91,2] = PR[GP1:90,2] + 46.068;
   1:L PR[91] 10mm/sec CNT100;
   1:  PR[GP1:91,1] = PR[GP1:90,1] + 6.487;
   1:  PR[GP1:91,2] = PR[GP1:90,2] + 48.407;
   1:L PR[91] 10mm/sec CNT100;
   1:  PR[GP1:91,1] = PR[GP1:90,1] + -0.265;
   1:  PR[GP1:91,2] = PR[GP1:90,2] + 49.669;
   1:L PR[91] 10mm/sec CNT100;
   1:  PR[GP1:91,1] = PR[GP1:90,1] + -7.015;
   1:  PR[GP1:91,2] = PR[GP1:90,2] + 48.406;
   1:L PR[91] 10mm/sec CNT100;
   1:  PR[GP1:91,1] = PR[GP1:90,1] + -18.768;
   1:  PR[GP1:91,2] = PR[GP1:90,2] + 46.068;
   1:L PR[91] 10mm/sec CNT100;
   1:  PR[GP1:91,1] = PR[GP1:90,1] + -24.603;
   1:  PR[GP1:91,2] = PR[GP1:90,2] + 42.454;
   1:L PR[91] 10mm/sec CNT100;
   1:  PR[GP1:91,1] = PR[GP1:90,1] + -34.580;
   1:  PR[GP1:91,2] = PR[GP1:90,2] + 35.788;
   1:L PR[91] 10mm/sec CNT100;
   1:  PR[GP1:91,1] = PR[GP1:90,1] + -37.857;
   1:  PR[GP1:91,2] = PR[GP1:90,2] + 31.841;
   1:L PR[91] 10mm/sec CNT100;
   1:  PR[GP1:91,1] = PR[GP1:90,1] + -44.530;
   1:  PR[GP1:91,2] = PR[GP1:90,2] + 21.853;
   1:L PR[91] 10mm/sec CNT100;
   1:  PR[GP1:91,1] = PR[GP1:90,1] + -46.595;
   1:  PR[GP1:91,2] = PR[GP1:90,2] + 17.175;
   1:L PR[91] 10mm/sec CNT100;
   1:  PR[GP1:91,1] = PR[GP1:90,1] + -47.311;
   1:  PR[GP1:91,2] = PR[GP1:90,2] + 12.042;
   1:L PR[91] 10mm/sec CNT100;
   1:  PR[GP1:91,1] = PR[GP1:90,1] + -49.655;
   1:  PR[GP1:91,2] = PR[GP1:90,2] + 0.261;
   1:L PR[91] 10mm/sec CNT100;
   1:  PR[GP1:91,1] = PR[GP1:90,1] + -48.946;
   1:  PR[GP1:91,2] = PR[GP1:90,2] + -4.820;
   1:L PR[91] 10mm/sec CNT100;
   1:  PR[GP1:91,1] = PR[GP1:90,1] + -46.602;
   1:  PR[GP1:91,2] = PR[GP1:90,2] + -16.601;
   1:L PR[91] 10mm/sec CNT100;
   1:  PR[GP1:91,1] = PR[GP1:90,1] + -44.530;
   1:  PR[GP1:91,2] = PR[GP1:90,2] + -21.295;
   1:L PR[91] 10mm/sec CNT100;
   1:  PR[GP1:91,1] = PR[GP1:90,1] + -37.857;
   1:  PR[GP1:91,2] = PR[GP1:90,2] + -31.283;
   1:L PR[91] 10mm/sec CNT100;
   1:  PR[GP1:91,1] = PR[GP1:90,1] + -34.580;
   1:  PR[GP1:91,2] = PR[GP1:90,2] + -35.230;
   1:L PR[91] 10mm/sec CNT100;
   1:  PR[GP1:91,1] = PR[GP1:90,1] + -24.603;
   1:  PR[GP1:91,2] = PR[GP1:90,2] + -41.896;
   1:L PR[91] 10mm/sec CNT100;
   1:  PR[GP1:91,1] = PR[GP1:90,1] + -18.771;
   1:  PR[GP1:91,2] = PR[GP1:90,2] + -45.508;
   1:L PR[91] 10mm/sec CNT100;
   1:  PR[GP1:91,1] = PR[GP1:90,1] + -12.014;
   1:  PR[GP1:91,2] = PR[GP1:90,2] + -46.772;
   1:L PR[91] 10mm/sec CNT100;
   1:  PR[GP1:91,1] = PR[GP1:90,1] + -0.261;
   1:  PR[GP1:91,2] = PR[GP1:90,2] + -49.110;
   1:L PR[91] 10mm/sec CNT100;
   1:  PR[GP1:91,1] = PR[GP1:90,1] + 5.386;
   1:  PR[GP1:91,2] = PR[GP1:90,2] + -48.054;
   1:  PR[GP1:91,3] = PR[GP1:90,3] + 135.115;
   1:L PR[91] 10mm/sec CNT100;
   1:  PR[GP1:91,1] = PR[GP1:90,1] + 18.306;
   1:  PR[GP1:91,2] = PR[GP1:90,2] + -45.484;
   1:L PR[91] 10mm/sec CNT100;
   1:  PR[GP1:91,1] = PR[GP1:90,1] + 23.190;
   1:  PR[GP1:91,2] = PR[GP1:90,2] + -42.459;
   1:L PR[91] 10mm/sec CNT100;
   1:  PR[GP1:91,1] = PR[GP1:90,1] + 34.155;
   1:  PR[GP1:91,2] = PR[GP1:90,2] + -35.133;
   1:L PR[91] 10mm/sec CNT100;
   1:  PR[GP1:91,1] = PR[GP1:90,1] + 36.894;
   1:  PR[GP1:91,2] = PR[GP1:90,2] + -31.834;
   1:L PR[91] 10mm/sec CNT100;
   1:  PR[GP1:91,1] = PR[GP1:90,1] + 44.228;
   1:  PR[GP1:91,2] = PR[GP1:90,2] + -20.856;
   1:L PR[91] 10mm/sec CNT100;
   1:  PR[GP1:91,1] = PR[GP1:90,1] + 45.953;
   1:  PR[GP1:91,2] = PR[GP1:90,2] + -16.950;
   1:L PR[91] 10mm/sec CNT100;
   1:  PR[GP1:91,1] = PR[GP1:90,1] + 46.553;
   1:  PR[GP1:91,2] = PR[GP1:90,2] + -12.651;
   1:L PR[91] 10mm/sec CNT100;
   1:  PR[GP1:91,1] = PR[GP1:90,1] + 49.129;
   1:  PR[GP1:91,2] = PR[GP1:90,2] + 0.297;
   1:L PR[91] 10mm/sec CNT100;
   1:  PR[GP1:91,1] = PR[GP1:90,1] + 48.536;
   1:  PR[GP1:91,2] = PR[GP1:90,2] + 4.543;
   1:L PR[91] 10mm/sec CNT100;
   1:  PR[GP1:91,1] = PR[GP1:90,1] + 45.960;
   1:  PR[GP1:91,2] = PR[GP1:90,2] + 17.492;
   1:L PR[91] 10mm/sec CNT100;
   1:  PR[GP1:91,1] = PR[GP1:90,1] + 44.228;
   1:  PR[GP1:91,2] = PR[GP1:90,2] + 21.414;
   1:L PR[91] 10mm/sec CNT100;
   1:  PR[GP1:91,1] = PR[GP1:90,1] + 36.894;
   1:  PR[GP1:91,2] = PR[GP1:90,2] + 32.392;
   1:L PR[91] 10mm/sec CNT100;
   1:  PR[GP1:91,1] = PR[GP1:90,1] + 34.155;
   1:  PR[GP1:91,2] = PR[GP1:90,2] + 35.691;
   1:L PR[91] 10mm/sec CNT100;
   1:  PR[GP1:91,1] = PR[GP1:90,1] + 23.190;
   1:  PR[GP1:91,2] = PR[GP1:90,2] + 43.017;
   1:L PR[91] 10mm/sec CNT100;
   1:  PR[GP1:91,1] = PR[GP1:90,1] + 18.306;
   1:  PR[GP1:91,2] = PR[GP1:90,2] + 46.042;
   1:L PR[91] 10mm/sec CNT100;
   1:  PR[GP1:91,1] = PR[GP1:90,1] + 5.386;
   1:  PR[GP1:91,2] = PR[GP1:90,2] + 48.612;
   1:L PR[91] 10mm/sec CNT100;
   1:  PR[GP1:91,1] = PR[GP1:90,1] + -0.264;
   1:  PR[GP1:91,2] = PR[GP1:90,2] + 49.669;
   1:L PR[91] 10mm/sec CNT100;
   1:  PR[GP1:91,1] = PR[GP1:90,1] + -5.913;
   1:  PR[GP1:91,2] = PR[GP1:90,2] + 48.612;
   1:L PR[91] 10mm/sec CNT100;
   1:  PR[GP1:91,1] = PR[GP1:90,1] + -18.833;
   1:  PR[GP1:91,2] = PR[GP1:90,2] + 46.042;
   1:L PR[91] 10mm/sec CNT100;
   1:  PR[GP1:91,1] = PR[GP1:90,1] + -23.715;
   1:  PR[GP1:91,2] = PR[GP1:90,2] + 43.018;
   1:L PR[91] 10mm/sec CNT100;
   1:  PR[GP1:91,1] = PR[GP1:90,1] + -34.682;
   1:  PR[GP1:91,2] = PR[GP1:90,2] + 35.691;
   1:L PR[91] 10mm/sec CNT100;
   1:  PR[GP1:91,1] = PR[GP1:90,1] + -37.420;
   1:  PR[GP1:91,2] = PR[GP1:90,2] + 32.392;
   1:L PR[91] 10mm/sec CNT100;
   1:  PR[GP1:91,1] = PR[GP1:90,1] + -44.755;
   1:  PR[GP1:91,2] = PR[GP1:90,2] + 21.415;
   1:L PR[91] 10mm/sec CNT100;
   1:  PR[GP1:91,1] = PR[GP1:90,1] + -46.479;
   1:  PR[GP1:91,2] = PR[GP1:90,2] + 17.508;
   1:L PR[91] 10mm/sec CNT100;
   1:  PR[GP1:91,1] = PR[GP1:90,1] + -47.079;
   1:  PR[GP1:91,2] = PR[GP1:90,2] + 13.209;
   1:L PR[91] 10mm/sec CNT100;
   1:  PR[GP1:91,1] = PR[GP1:90,1] + -49.655;
   1:  PR[GP1:91,2] = PR[GP1:90,2] + 0.261;
   1:L PR[91] 10mm/sec CNT100;
   1:  PR[GP1:91,1] = PR[GP1:90,1] + -49.063;
   1:  PR[GP1:91,2] = PR[GP1:90,2] + -3.985;
   1:L PR[91] 10mm/sec CNT100;
   1:  PR[GP1:91,1] = PR[GP1:90,1] + -46.486;
   1:  PR[GP1:91,2] = PR[GP1:90,2] + -16.934;
   1:L PR[91] 10mm/sec CNT100;
   1:  PR[GP1:91,1] = PR[GP1:90,1] + -44.755;
   1:  PR[GP1:91,2] = PR[GP1:90,2] + -20.857;
   1:L PR[91] 10mm/sec CNT100;
   1:  PR[GP1:91,1] = PR[GP1:90,1] + -37.420;
   1:  PR[GP1:91,2] = PR[GP1:90,2] + -31.834;
   1:L PR[91] 10mm/sec CNT100;
   1:  PR[GP1:91,1] = PR[GP1:90,1] + -34.682;
   1:  PR[GP1:91,2] = PR[GP1:90,2] + -35.133;
   1:L PR[91] 10mm/sec CNT100;
   1:  PR[GP1:91,1] = PR[GP1:90,1] + -23.715;
   1:  PR[GP1:91,2] = PR[GP1:90,2] + -42.460;
   1:L PR[91] 10mm/sec CNT100;
   1:  PR[GP1:91,1] = PR[GP1:90,1] + -18.836;
   1:  PR[GP1:91,2] = PR[GP1:90,2] + -45.482;
   1:L PR[91] 10mm/sec CNT100;
   1:  PR[GP1:91,1] = PR[GP1:90,1] + -13.181;
   1:  PR[GP1:91,2] = PR[GP1:90,2] + -46.539;
   1:L PR[91] 10mm/sec CNT100;
   1:  PR[GP1:91,1] = PR[GP1:90,1] + -0.261;
   1:  PR[GP1:91,2] = PR[GP1:90,2] + -49.110;
   1:L PR[91] 10mm/sec CNT100;
   1:  PR[GP1:91,1] = PR[GP1:90,1] + 4.284;
   1:  PR[GP1:91,2] = PR[GP1:90,2] + -48.260;
